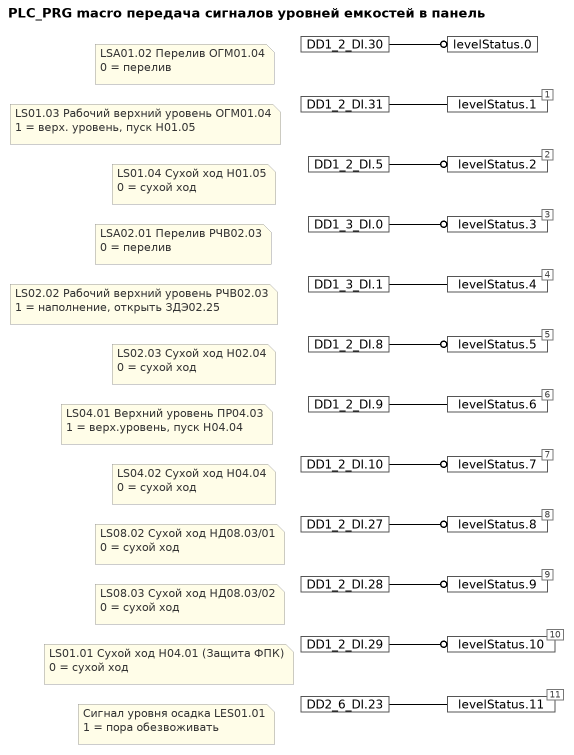
[picture p24: PLC_PRG macro передача сигналов уровней емкостей в панель (CFC)]
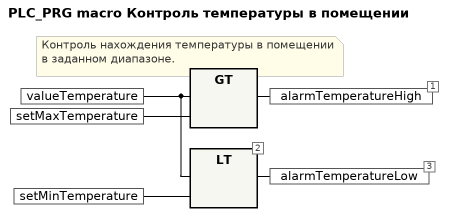
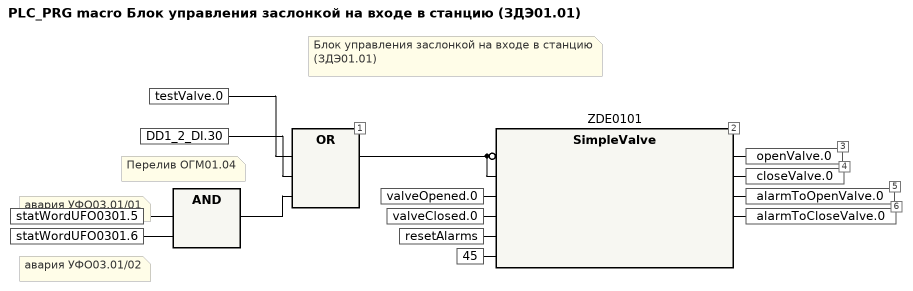
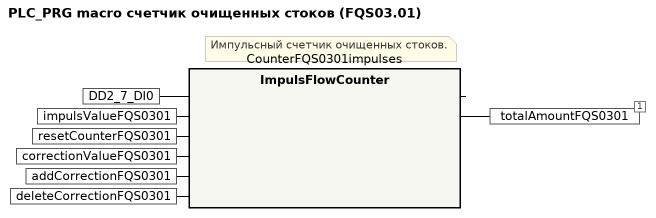
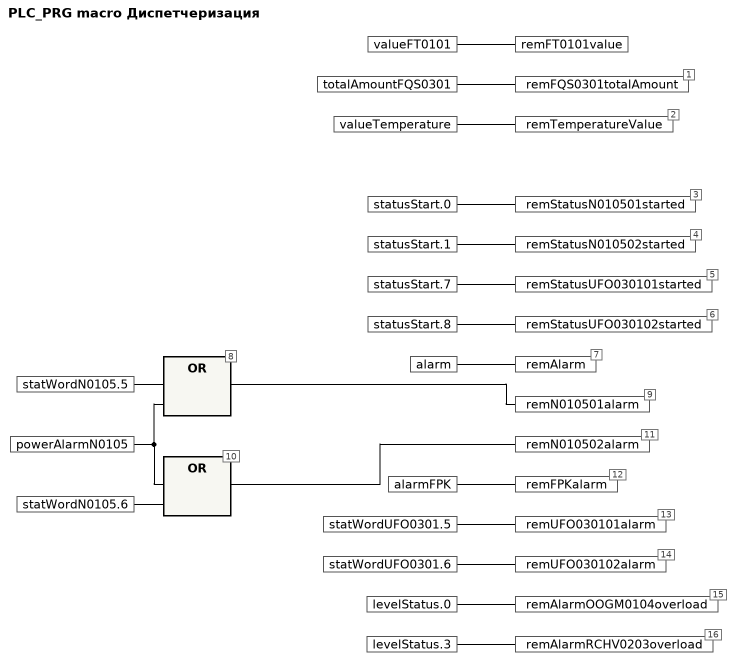
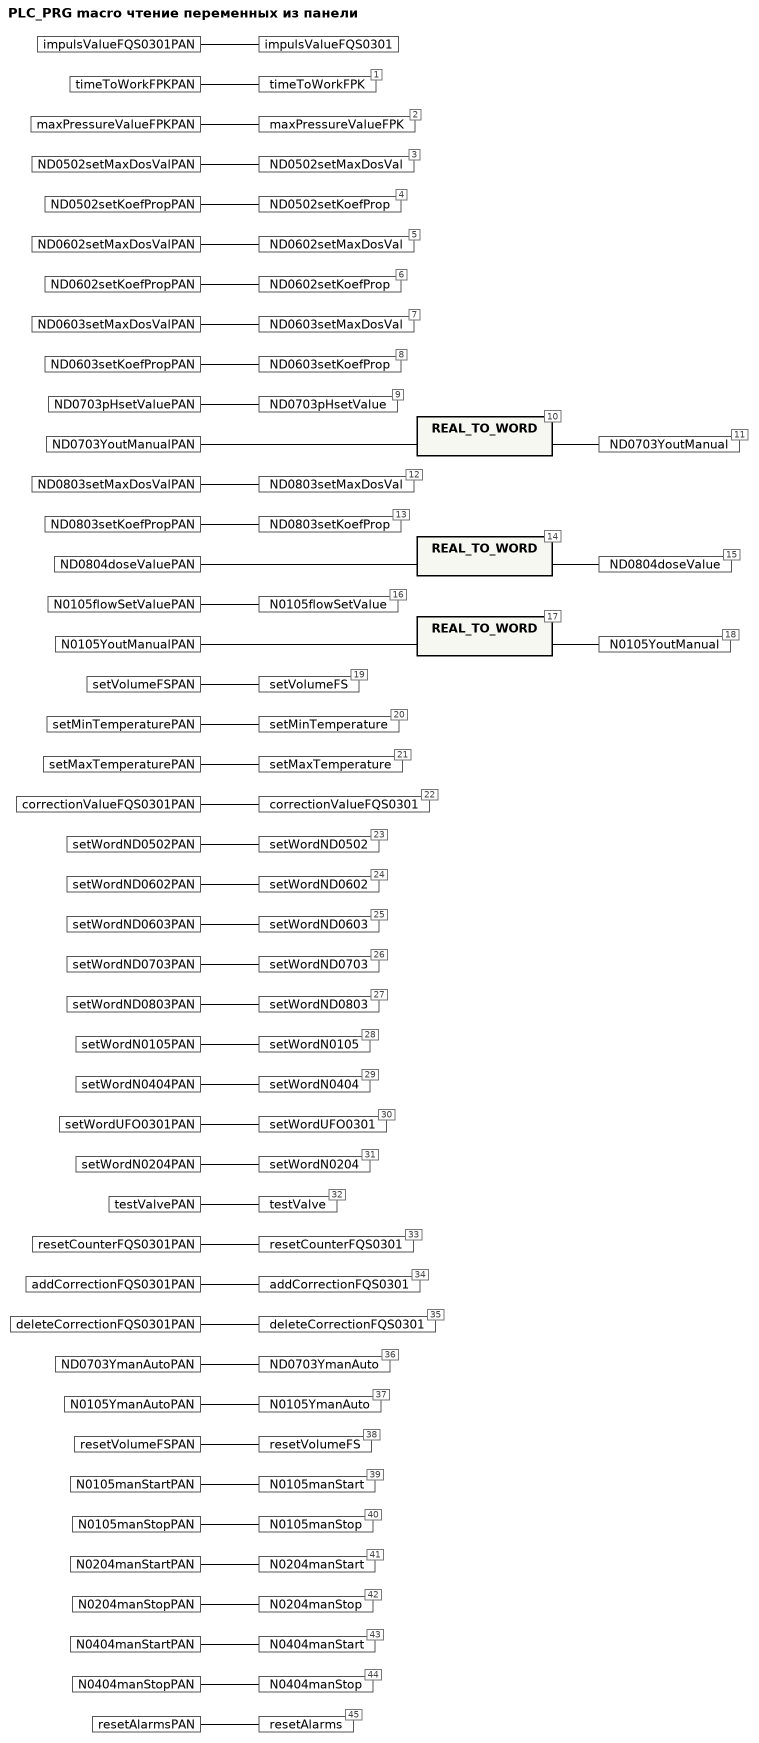
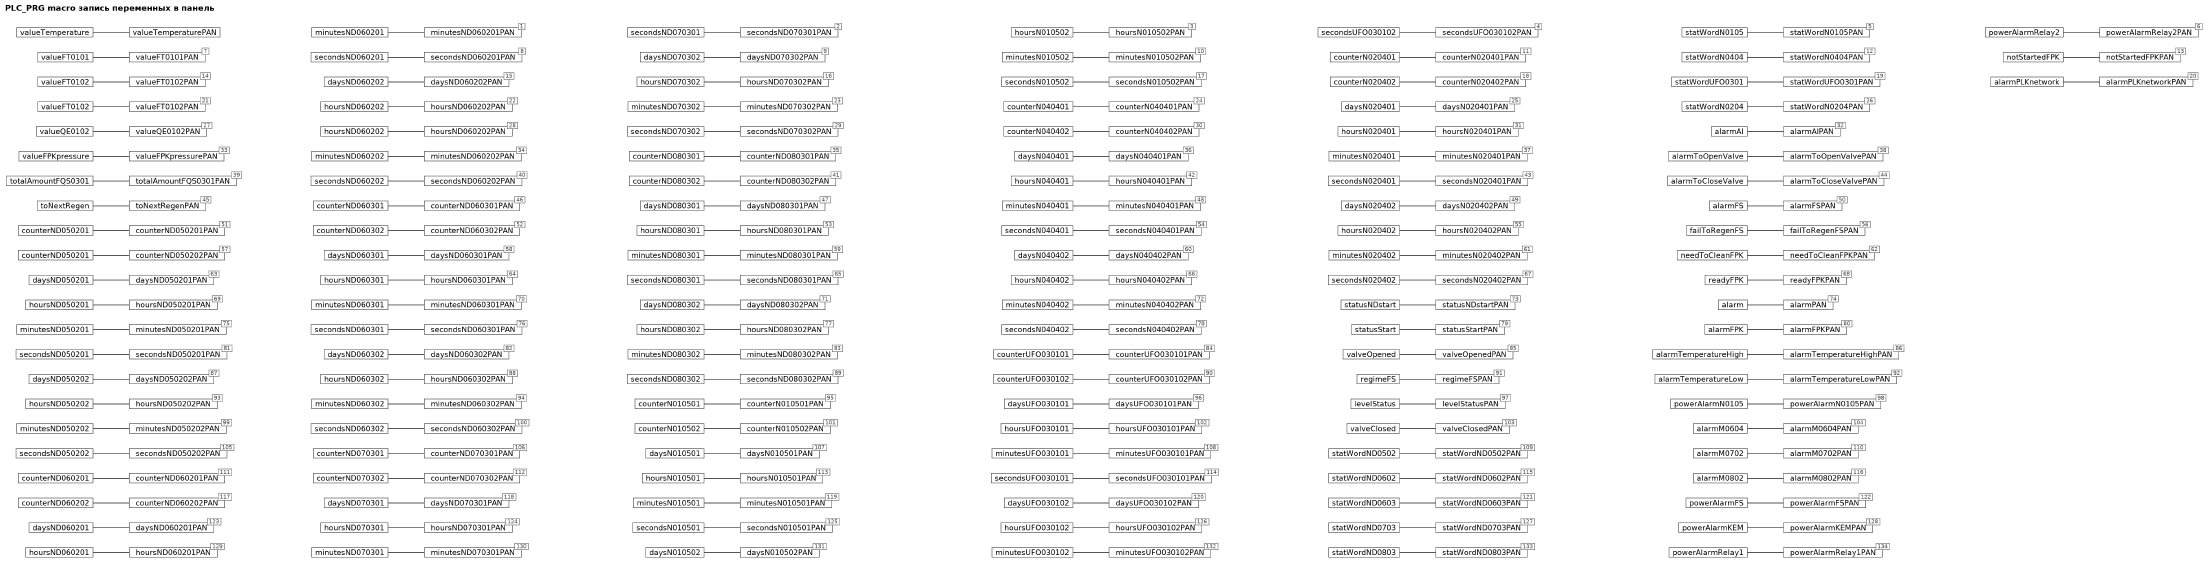
_CFC_ (* Continuous Function Chart, elements in execution order *)
#0 MACRO Блок задания всем режима по количеству включений при подаче питания()
	(* задать режим запуска УФО03.01 / по количеству включений *)
	(* задать режим запуска Н01.05 / по количеству включений *)
	(* задать режим запуска НД06.03 / по количеству включений *)
	(* задать режим запуска НД06.02 / по количеству включений *)
	(* задать режим запуска НД05.02 / по количеству включений *)
	(* задать режим запуска НД07.03 / по количеству включений *)
	(* задать режим запуска НД08.03 / по количеству включений *)
	(* задать режим запуска Н02.04 / по количеству включений *)
	(* задать режим запуска Н04.04 / по количеству включений *)
	#1 StartInitiBlock:R_TRIG(CLK: TRUE)
	#2 startInitializer <= #1.Q
	#3 setWordND0502.3 <= #1.Q
	#4 setWordND0602.3 <= #1.Q
	#5 setWordND0603.3 <= #1.Q
	#6 setWordND0703.3 <= #1.Q
	#7 setWordND0803.3 <= #1.Q
	#8 setWordN0105.3 <= #1.Q
	#9 setWordN0204.3 <= #1.Q
	#10 setWordN0404.3 <= #1.Q
	#11 setWordUFO0301.3 <= #1.Q
END_MACRO
#12 MACRO Управление доз.насосами НД05.02/01 и НД05.02/02()
	(* Управление доз.насосами НД05.02/01 и НД05.02/02 / пропорционально расходу по показаниям расходомера FT01.01 *)
	(* управление НД05.02/02 = 4...20мА *)
	(* управление НД05.02/01 = 4...20мА *)
	(* Если на входе sel = true, то нижнее значение, / иначе - посередине. Для того, чтобы при / выключении насоса не висело задание, / а сбрасывалось в ноль. *)
	(* Пуск НД05.02/01 *)
	(* Пуск НД05.02/02 *)
	#13 ND0502dosing:DosingPumpProportional(valueFT0101, -, ND0502setMaxDosVal, -, -, ND0502setKoefProp, -)
	#14 statWordND0502.0 <= #13.out 2
	#15 setWordND0502.0 <= #13.out 3
	#16 REAL_TO_WORD(#13.out 1)
	#17 ND0502manager:RichTwoPumpManager(setWordND0502.0, setWordND0502.1, setWordND0502.2, setWordND0502.3, setWordND0502.4, setWordND0502.5, setWordND0502.6, setWordND0502.7, setWordND0502.8, setWordND0502.9, setWordND0502.10, setWordND0502.11, resetAlarms, -, alarmND.0, alarmND.1)
	#18 statWordND0502.1 <= #17.out 1
	#19 statWordND0502.2 <= #17.out 2
	#20 statWordND0502.3 <= #17.out 3
	#21 statWordND0502.4 <= #17.out 4
	#22 counterND050201 <= #17.out 5
	#23 counterND050202 <= #17.out 6
	#24 daysND050201 <= #17.out 7
	#25 hoursND050201 <= #17.out 8
	#26 minutesND050201 <= #17.out 9
	#27 secondsND050201 <= #17.out 10
	#28 daysND050202 <= #17.out 11
	#29 hoursND050202 <= #17.out 12
	#30 minutesND050202 <= #17.out 13
	#31 secondsND050202 <= #17.out 14
	#32 statusNDstart.0 <= #17.out 15
	#33 DD1_1_DO.12 <= #17.out 15
	#34 DD1_1_DO.13 <= #17.out 16
	#35 statusNDstart.1 <= #17.out 16
	#36 statWordND0502.5 <= #17.out 19
	#37 statWordND0502.6 <= #17.out 20
	#38 SEL(#17.out 15, 4, #16)
	#39 lintrafoND050201:LIN_TRAFO(IN: #38, IN_MIN: 4, IN_MAX: 20, OUT_MIN: 0, OUT_MAX: 1000)
	#40 REAL_TO_WORD(#39.OUT)
	#41 DD1_4_AO0 <= #40
	#42 SEL(#17.out 16, 4, #16)
	#43 lintrafoND050202:LIN_TRAFO(IN: #42, IN_MIN: 4, IN_MAX: 20, OUT_MIN: 0, OUT_MAX: 1000)
	#44 REAL_TO_WORD(#43.OUT)
	#45 DD1_4_AO1 <= #44
END_MACRO
#46 MACRO Управление насосами Н01.05/01 и Н01.05/02()
	(* статус старт Н01.05/02 *)
	(* статус старт Н01.05/01 *)
	(* производительность для ЧРП Н01.05 *)
	(* командное слово для ЧРП Н01.05 *)
	(* Рабочий верхний уровень ОГМ01.04 *)
	(* Перелив ОГМ01.04 *)
	(* Сухой ход Н01.05 *)
	(* Термоконтакт Н01.05/02 *)
	(* Термоконтакт Н01.05/01 *)
	(* Авария привода Н01.05 (сигнал авария от ЧРП А1) *)
	(* Сигнал - ЧРП в режиме ПУСК, один из насосов работает. / Сигнал на лампы HL3-4 через доп.контакты КМ3.2 и КМ4.2 *)
	(* Питание Н01.05/01 (КМ4) *)
	(* Питание Н01.05/01 (КМ3) *)
	(* регулируем от 30 до 50Гц, чтобы не перегреть двигатель / 30Гц = 3258 *)
	(* 5430 = 50Гц *)
	(* Работа Н01.05 / Поддержание заданного расхода по FT01.02 / Пуск по верхнему рабочему уровню (LS01.03) или вручную с пульта / стоп по защите от сухого хода (LS01.04) или вручную с пульта *)
	(* Питание ЧРП Н01.05 (КМ2) *)
	(* слово состояния для ЧРП Н01.05 / сигнал - авария *)
	#47 linTrafoN0105:LIN_TRAFO(IN: N0105YoutManual, IN_MIN: 0, IN_MAX: 100, OUT_MIN: 0, OUT_MAX: 5430)
	#48 PID_ND0105:PID(ACTUAL: valueFT0102, SET_POINT: N0105flowSetValue, KP: 1, TN: 10, TV: 1, Y_MANUAL: #47.OUT, Y_OFFSET: 0, Y_MIN: 0, Y_MAX: 5430, MANUAL: N0105YmanAuto, RESET: #48.OVERFLOW)
	#49 LT(#48.Y, 3258)
	#50 SEL(#49, #48.Y, 3258)
	#51 REAL_TO_WORD(#50)
	#52 zad_rsN0105 <= #51
	#53 OR(DD1_2_DI.31, NOT DD1_2_DI.30, N0105manStart)
	#54 OR(NOT DD1_2_DI.5, N0105manStop)
	#55 rsTrigN0105:RS(SET: #53, RESET1: #54)
	#56 setWordN0105.0 <= #55.Q1
	#57 OR(DD1_2_DI.0, stat_wordN0105.3)
	#58 ND0105manager:TwoPumpOneDriveManager(setWordN0105.0, setWordN0105.1, setWordN0105.2, setWordN0105.3, setWordN0105.4, setWordN0105.5, setWordN0105.6, setWordN0105.7, setWordN0105.8, setWordN0105.9, setWordN0105.10, setWordN0105.11, resetAlarms, -, NOT DD1_2_DI.3, NOT DD1_2_DI.4, #57)
	#59 statWordN0105.1 <= #58.out 1
	#60 statWordN0105.2 <= #58.out 2
	#61 statWordN0105.3 <= #58.out 3
	#62 statWordN0105.4 <= #58.out 4
	#63 counterN010501 <= #58.out 5
	#64 counterN010502 <= #58.out 6
	#65 daysN010501 <= #58.out 7
	#66 hoursN010501 <= #58.out 8
	#67 minutesN010501 <= #58.out 9
	#68 secondsN010501 <= #58.out 10
	#69 daysN010502 <= #58.out 11
	#70 hoursN010502 <= #58.out 12
	#71 minutesN010502 <= #58.out 13
	#72 secondsN010502 <= #58.out 14
	#73 DD1_1_DO.0 <= #58.out 15
	#74 DD1_1_DO.1 <= #58.out 16
	#75 DD1_1_DO.2 <= #58.out 17
	#76 statWordN0105.5 <= #58.out 21
	#77 statWordN0105.6 <= #58.out 22
	#78 DD1_1_DO.3 <= #58.out 18
	#79 AND(DD1_1_DO.1, #58.out 18)
	#80 statusStart.0 <= #79
	#81 AND(#58.out 18, DD1_1_DO.2)
	#82 statusStart.1 <= #81
	#83 StartStopND0105:StartStopVFD(startStop: #58.out 18)
	#84 com_wordN0105 <= #83.commandWord
END_MACRO
#85 MACRO Сигналы "АВАРИЯ" от дозирующих насосов()
	(* Авария НД08.03/02 = stat_wordND080302.3 *)
	(* Авария НД08.03/01 = stat_wordND080301.3 *)
	(* Сигнал авария от физических выходов доз.насосов взят НЗ, т.е. / при замкнутом состоянии аварии нет. Если сигнал выдается только НО / (замкнуто = авария) - убрать инверсию здесь. / Сигнал авария по модбасу здесь взят как НО / т.е. false = норма, true - авария. *)
	(* Авария НД05.02/01 *)
	(* Авария НД05.02/02 *)
	(* Авария НД06.02/01 *)
	(* Авария НД06.02/02 *)
	(* Авария НД06.03/01 *)
	(* Авария НД06.03/02 *)
	(* Авария НД07.03/01 *)
	(* Авария НД07.03/02 *)
	(* Авария НД08.04 *)
	#86 alarmND.0 <= NOT DD1_2_DI.18
	#87 alarmND.1 <= NOT DD1_2_DI.19
	#88 alarmND.2 <= NOT DD1_2_DI.20
	#89 alarmND.3 <= NOT DD1_2_DI.21
	#90 alarmND.4 <= NOT DD1_2_DI.22
	#91 alarmND.5 <= NOT DD1_2_DI.23
	#92 alarmND.6 <= NOT DD1_2_DI.24
	#93 alarmND.7 <= NOT DD1_2_DI.25
	#94 alarmND.8 <= NOT DD2_6_DI.22
END_MACRO
#95 MACRO Управление доз.насосами НД06.02/01 и НД06.02/02()
	(* Управление доз.насосами НД06.02/01 и НД06.02/02 / пропорционально расходу по показаниям расходомера FT01.02 *)
	(* управление НД06.02/02 = 4...20мА *)
	(* управление НД06.02/01 = 4...20мА *)
	(* Если на входе sel = true, то нижнее значение, / иначе - посередине. Для того, чтобы при / выключении насоса не висело задание, / а сбрасывалось в ноль. *)
	(* Пуск НД06.02/01 *)
	(* Пуск НД06.02/02 *)
	#96 ND0602dosing:DosingPumpProportional(valueFT0102, -, ND0602setMaxDosVal, -, -, ND0602setKoefProp, -)
	#97 statWordND0602.0 <= #96.out 2
	#98 setWordND0602.0 <= #96.out 3
	#99 REAL_TO_WORD(#96.out 1)
	#100 ND0602manager:RichTwoPumpManager(setWordND0602.0, setWordND0602.1, setWordND0602.2, setWordND0602.3, setWordND0602.4, setWordND0602.5, setWordND0602.6, setWordND0602.7, setWordND0602.8, setWordND0602.9, setWordND0602.10, setWordND0602.11, resetAlarms, -, alarmND.2, alarmND.3)
	#101 statWordND0602.1 <= #100.out 1
	#102 statWordND0602.2 <= #100.out 2
	#103 statWordND0602.3 <= #100.out 3
	#104 statWordND0602.4 <= #100.out 4
	#105 counterND060201 <= #100.out 5
	#106 counterND060202 <= #100.out 6
	#107 daysND060201 <= #100.out 7
	#108 hoursND060201 <= #100.out 8
	#109 minutesND060201 <= #100.out 9
	#110 secondsND060201 <= #100.out 10
	#111 daysND060202 <= #100.out 11
	#112 hoursND060202 <= #100.out 12
	#113 minutesND060202 <= #100.out 13
	#114 secondsND060202 <= #100.out 14
	#115 statusNDstart.2 <= #100.out 15
	#116 DD1_1_DO.14 <= #100.out 15
	#117 DD1_1_DO.15 <= #100.out 16
	#118 statusNDstart.3 <= #100.out 16
	#119 statWordND0602.5 <= #100.out 19
	#120 statWordND0602.6 <= #100.out 20
	#121 SEL(#100.out 15, 4, #99)
	#122 lintrafoND060201:LIN_TRAFO(IN: #121, IN_MIN: 4, IN_MAX: 20, OUT_MIN: 0, OUT_MAX: 1000)
	#123 REAL_TO_WORD(#122.OUT)
	#124 DD1_4_AO2 <= #123
	#125 SEL(#100.out 16, 4, #99)
	#126 lintrafoND060202:LIN_TRAFO(IN: #125, IN_MIN: 4, IN_MAX: 20, OUT_MIN: 0, OUT_MAX: 1000)
	#127 REAL_TO_WORD(#126.OUT)
	#128 DD1_4_AO3 <= #127
END_MACRO
#129 MACRO Блок управления насосами Н02.04/01 и Н02.04/02()
	(* Минимум один из фильтров в режиме промывки *)
	(* Пуск Н02.04/02 *)
	(* Открыт минимум один из клапанов КЭМ *)
	(* Сухой ход Н02.04 / 1 = норма / 0 = сухой ход *)
	(* Авария Н02.04/02 *)
	(* Авария Н02.04/01 *)
	(* Пуск Н02.04/01 *)
	(* Блок управления насосами Н02.04/01 и Н02.04/02 / Включен, если хоть один из клапанов КЭМ открыт, / один из фильтров в промывке старт/стоп вручную (тест). *)
	(* автоматический пуск/стоп *)
	(* ручной пуск/стоп с защитой от сухого хода *)
	(* Сигнал на запуск насоса / согласно выбранному режиму *)
	#130 WORD_TO_BOOL(openedKEM)
	#131 WORD_TO_BOOL(regimeFS)
	#132 OR(#130, #131)
	#133 AND(#132, DD1_2_DI.8)
	#134 OR(NOT DD1_2_DI.8, N0204manStop)
	#135 N0204startTrig:RS(SET: N0204manStart, RESET1: #134)
	#136 OR(#133, #135.Q1)
	#137 setWordN0204.0 <= #136
	#138 N0204manager:RichTwoPumpManager(setWordN0204.0, setWordN0204.1, setWordN0204.2, setWordN0204.3, setWordN0204.4, setWordN0204.5, setWordN0204.6, setWordN0204.7, setWordN0204.8, setWordN0204.9, setWordN0204.10, setWordN0204.11, resetAlarms, -, DD1_2_DI.6, DD1_2_DI.7)
	#139 statWordN0204.1 <= #138.out 1
	#140 statWordN0204.2 <= #138.out 2
	#141 statWordN0204.3 <= #138.out 3
	#142 statWordN0204.4 <= #138.out 4
	#143 counterN020401 <= #138.out 5
	#144 counterN020402 <= #138.out 6
	#145 daysN020401 <= #138.out 7
	#146 hoursN020401 <= #138.out 8
	#147 minutesN020401 <= #138.out 9
	#148 daysN020402 <= #138.out 11
	#149 hoursN020402 <= #138.out 12
	#150 minutesN020402 <= #138.out 13
	#151 statusStart.2 <= #138.out 15
	#152 secondsN020402 <= #138.out 14
	#153 DD1_1_DO.4 <= #138.out 15
	#154 DD1_1_DO.5 <= #138.out 16
	#155 statusStart.3 <= #138.out 16
	#156 statWordN0204.5 <= #138.out 19
	#157 statWordN0204.6 <= #138.out 20
END_MACRO
#158 MACRO Блок сбора всех аварий и выдачи одной общей()
	(* Контроль состояния сети ПЛК, задержка выдачи сигнала = 20 сек. / Контроль обрыва в сети (модуль отсоединен, или модуль в аварии. *)
	(* ошибка блоков дозирования / (неправильно выставлены / параметры в настройках) *)
	(* лампа Авария / (щит-1) *)
	(* Авария питания ЧРП А1 (автомат ЧРП выключен) *)
	(* Перелив ОГМ01.04 (отстойник) *)
	(* Перелив РЧВ02.03 *)
	(* Авария М08.02 (УПФ) *)
	(* Авария М07.02 (УПЩ) *)
	(* Авария М06.04 (УПК) *)
	(* Авария питания управляющих клапанов фильтров *)
	(* Авария питания клапанов КЭМ *)
	(* Авария питания K, KM, HL щит1 *)
	(* Авария питания реле щита 2 *)
	(* Авария фильтр-пресса (ФП) *)
	#159 WORD_TO_BOOL(alarmAI)
	#160 DWORD_TO_BOOL(alarmToOpenValve)
	#161 DWORD_TO_BOOL(alarmToCloseValve)
	#162 WORD_TO_BOOL(alarmFS)
	#163 WORD_TO_BOOL(failToRegenFS)
	#164 EQ(lastError, 0)
	#165 alarmPLKnetworkDelay:TOF(IN: #164, PT: T#20s)
	#166 NOT(#165.Q)
	#167 alarmPLKnetwork <= #166
	#168 OR(#159, alarmTemperatureHigh, alarmTemperatureLow, statWordND0502.5, statWordND0502.6, statWordND0602.5, statWordND0602.6, statWordND0603.5, statWordND0603.6, statWordND0703.5, statWordND0703.6, statWordND0803.5, statWordND0803.6, powerAlarmN0105, statWordN0105.5, statWordN0105.6, levelStatus.0, statWordN0204.5, statWordN0204.6, statWordN0404.5, statWordN0404.6, #160, #161, alarmM0604, alarmM0702, alarmM0802, powerAlarmFS, levelStatus.3, powerAlarmKEM, powerAlarmRelay1, powerAlarmRelay2, alarmFPK, notStartedFPK, #162, #163, statWordUFO0301.5, statWordUFO0301.6, statWordND0502.0, statWordND0602.0, statWordND0603.0, statWordND0803.0, alarmND.8, #166)
	#169 alarm <= #168
	#170 DD1_1_DO.8 <= #168
	#171 powerAlarmN0105 <= DD1_2_DI.2
	#172 alarmM0604 <= NOT DD1_2_DI.15
	#173 alarmM0702 <= NOT DD1_2_DI.16
	#174 alarmM0802 <= NOT DD1_2_DI.17
	#175 powerAlarmFS <= NOT DD1_2_DI.26
	#176 powerAlarmKEM <= NOT DD1_3_DI.2
	#177 powerAlarmRelay1 <= NOT DD1_2_DI.1
	#178 powerAlarmRelay2 <= NOT DD2_4_DI.0
	#179 alarmFPK <= DD2_6_DI.21
END_MACRO
#180 MACRO Управление доз.насосами НД06.03/01 и НД06.03/02()
	(* Управление доз.насосами НД06.03/01 и НД06.03/02 / пропорционально расходу по показаниям расходомера FT01.01 *)
	(* управление НД06.03/02 = 4...20мА *)
	(* управление НД06.03/01 = 4...20мА *)
	(* Если на входе sel = true, то нижнее значение, / иначе - посередине. Для того, чтобы при / выключении насоса не висело задание, / а сбрасывалось в ноль. *)
	(* Пуск НД06.03/01 *)
	(* Пуск НД06.03/02 *)
	#181 ND0603dosing:DosingPumpProportional(valueFT0101, -, ND0603setMaxDosVal, -, -, ND0603setKoefProp, -)
	#182 statWordND0603.0 <= #181.out 2
	#183 setWordND0603.0 <= #181.out 3
	#184 REAL_TO_WORD(#181.out 1)
	#185 ND0603manager:RichTwoPumpManager(setWordND0603.0, setWordND0603.1, setWordND0603.2, setWordND0603.3, setWordND0603.4, setWordND0603.5, setWordND0603.6, setWordND0603.7, setWordND0603.8, setWordND0603.9, setWordND0603.10, setWordND0603.11, resetAlarms, -, alarmND.4, alarmND.5)
	#186 statWordND0603.1 <= #185.out 1
	#187 statWordND0603.2 <= #185.out 2
	#188 statWordND0603.3 <= #185.out 3
	#189 statWordND0603.4 <= #185.out 4
	#190 counterND060301 <= #185.out 5
	#191 counterND060302 <= #185.out 6
	#192 daysND060301 <= #185.out 7
	#193 hoursND060301 <= #185.out 8
	#194 minutesND060301 <= #185.out 9
	#195 secondsND060301 <= #185.out 10
	#196 daysND060302 <= #185.out 11
	#197 hoursND060302 <= #185.out 12
	#198 minutesND060302 <= #185.out 13
	#199 secondsND060302 <= #185.out 14
	#200 statusNDstart.4 <= #185.out 15
	#201 DD1_1_DO.16 <= #185.out 15
	#202 DD1_1_DO.17 <= #185.out 16
	#203 statusNDstart.5 <= #185.out 16
	#204 statWordND0603.5 <= #185.out 19
	#205 statWordND0603.6 <= #185.out 20
	#206 SEL(#185.out 15, 4, #184)
	#207 linrtafoND060301:LIN_TRAFO(IN: #206, IN_MIN: 4, IN_MAX: 20, OUT_MIN: 0, OUT_MAX: 1000)
	#208 REAL_TO_WORD(#207.OUT)
	#209 DD1_4_AO4 <= #208
	#210 SEL(#185.out 16, 4, #184)
	#211 linrtafoND060302:LIN_TRAFO(IN: #210, IN_MIN: 4, IN_MAX: 20, OUT_MIN: 0, OUT_MAX: 1000)
	#212 REAL_TO_WORD(#211.OUT)
	#213 DD1_4_AO5 <= #212
END_MACRO
#214 MACRO Блок управления насосами Н04.04/01 и Н04.04/02()
	(* Сухой ход Н04.04 / 1 = норма / 0 = сухой ход *)
	(* Блок управления насосами Н04.04/01 и Н04.04/02 / Дренажные насосы. Работа по поплавкам (LS04.01 и LS04.02) или пуск вручную (тест). *)
	(* автоматический пуск/стоп *)
	(* ручной пуск/стоп с защитой от сухого хода *)
	(* Сигнал на запуск насоса / согласно выбранному режиму *)
	(* Пуск Н04.04/01 *)
	(* Пуск Н04.04/02 *)
	(* Верхний уровень ПР04.03 *)
	(* Авария Н04.04/01 *)
	(* Авария Н04.04/02 *)
	#215 AND(DD1_2_DI.9, DD1_2_DI.10)
	#216 OR(NOT DD1_2_DI.10, N0404manStop)
	#217 N0404startTrig:RS(SET: N0404manStart, RESET1: #216)
	#218 OR(#215, #217.Q1)
	#219 setWordN0404.0 <= #218
	#220 N0404manager:RichTwoPumpManager(setWordN0404.0, setWordN0404.1, setWordN0404.2, setWordN0404.3, setWordN0404.4, setWordN0404.5, setWordN0404.6, setWordN0404.7, setWordN0404.8, setWordN0404.9, setWordN0404.10, setWordN0404.11, resetAlarms, -, DD1_2_DI.11, DD1_2_DI.12)
	#221 statWordN0404.1 <= #220.out 1
	#222 statWordN0404.2 <= #220.out 2
	#223 statWordN0404.3 <= #220.out 3
	#224 statWordN0404.4 <= #220.out 4
	#225 counterN040401 <= #220.out 5
	#226 counterN040402 <= #220.out 6
	#227 daysN040401 <= #220.out 7
	#228 hoursN040401 <= #220.out 8
	#229 minutesN040401 <= #220.out 9
	#230 secondsN040401 <= #220.out 10
	#231 daysN040402 <= #220.out 11
	#232 hoursN040402 <= #220.out 12
	#233 minutesN040402 <= #220.out 13
	#234 DD1_1_DO.6 <= #220.out 15
	#235 secondsN040402 <= #220.out 14
	#236 statusStart.4 <= #220.out 15
	#237 statusStart.5 <= #220.out 16
	#238 DD1_1_DO.7 <= #220.out 16
	#239 statWordN0404.5 <= #220.out 19
	#240 statWordN0404.6 <= #220.out 20
END_MACRO
#241 MACRO AI PLC (блок обработки аналоговых входов)()
	(* Здесь принимаем сигнал от входа ПЛК, в нем должно быть выставлен диапазон 0...20 / Задаем максимальное и минимальное значение для измеряемой величины при 4 и 20мА на датчике. *)
	(* рН *)
	(* рН *)
	(* бар *)
	(* куб.м./час *)
	(* куб.м./час *)
	(* Давление на входе / в фильтр-пресс *)
	(* рН-ОВП метр QE01.02 *)
	(* рН-ОВП метр QE01.01 *)
	(* Расходомер FT01.02 *)
	(* град.С *)
	(* Расходомер FT01.01 *)
	(* датчик температуры / в помещении TT01 *)
	(* Авария датчика температуры *)
	(* Авария расходомера FT01.01 *)
	(* Авария расходомера FT01.02 *)
	(* Авария рН-метра QE01.01 *)
	(* Авария рН-метра QE01.02 *)
	(* Авария входа приема показаний / давления на входе в фильтр *)
	#242 ControlAI0:ControlAI(DD2_7_AI0, -40, 80)
	#243 valueTemperature <= #242.out 1
	#244 alarmAI.0 <= #242.out 2
	#245 ControlAI1:ControlAI(DD2_7_AI1, -, 600)
	#246 valueFT0101 <= #245.out 1
	#247 alarmAI.1 <= #245.out 2
	#248 ControlAI2:ControlAI(DD2_7_AI2, -, 600)
	#249 valueFT0102 <= #248.out 1
	#250 alarmAI.2 <= #248.out 2
	#251 ControlAI3:ControlAI(DD2_7_AI3, -, 14)
	#252 valueQE0101 <= #251.out 1
	#253 alarmAI.3 <= #251.out 2
	#254 ControlAI4:ControlAI(DD2_7_AI4, -, 14)
	#255 valueQE0102 <= #254.out 1
	#256 alarmAI.4 <= #254.out 2
	#257 ControlAI5:ControlAI(DD2_7_AI5, -, 16)
	#258 valueFPKpressure <= #257.out 1
	#259 alarmAI.5 <= #257.out 2
END_MACRO
#260 MACRO Управление доз.насосами НД07.03/01 и НД07.03/02()
	(* коэф. P *)
	(* Пуск, если по FT01.01 / расход >= 10 куб.метров *)
	(* Управление доз.насосами НД07.03/01 и НД07.03/02 / поддержание заданного уровня рН по показаниям QE01.01 *)
	(* управление НД07.03/02 = 4...20мА *)
	(* управление НД07.03/01 = 4...20мА *)
	(* Если на входе sel = true, то нижнее значение, / иначе - посередине. Для того, чтобы при / выключении насоса не висело задание, / а сбрасывалось в ноль. *)
	(* Пуск НД07.03/01 *)
	(* Пуск НД07.03/02 *)
	(* коэф. I *)
	(* коэф. D *)
	(* Y при аварии *)
	#261 manYoutND0703:LIN_TRAFO(IN: ND0703YoutManual, IN_MIN: 0, IN_MAX: 100, OUT_MIN: 4, OUT_MAX: 20)
	#262 ND0703pidReg:PID(ACTUAL: valueQE0101, SET_POINT: ND0703pHsetValue, KP: 1, TN: 10, TV: 1, Y_MANUAL: #261.OUT, Y_OFFSET: 12, Y_MIN: 4, Y_MAX: 20, MANUAL: ND0703YmanAuto, RESET: #262.OVERFLOW)
	#263 REAL_TO_WORD(#262.Y)
	#264 GE(valueFT0101, 10)
	#265 ND0703manager:RichTwoPumpManager(#264, setWordND0703.1, setWordND0703.2, setWordND0703.3, setWordND0703.4, setWordND0703.5, setWordND0703.6, setWordND0703.7, setWordND0703.8, setWordND0703.9, setWordND0703.10, setWordND0703.11, resetAlarms, -, alarmND.6, alarmND.7)
	#266 statWordND0703.1 <= #265.out 1
	#267 statWordND0703.2 <= #265.out 2
	#268 statWordND0703.3 <= #265.out 3
	#269 statWordND0703.4 <= #265.out 4
	#270 counterND070301 <= #265.out 5
	#271 counterND070302 <= #265.out 6
	#272 daysND070301 <= #265.out 7
	#273 hoursND070301 <= #265.out 8
	#274 minutesND070301 <= #265.out 9
	#275 secondsND070301 <= #265.out 10
	#276 daysND070302 <= #265.out 11
	#277 hoursND070302 <= #265.out 12
	#278 minutesND070302 <= #265.out 13
	#279 secondsND070302 <= #265.out 14
	#280 statusNDstart.6 <= #265.out 15
	#281 DD1_1_DO.18 <= #265.out 15
	#282 DD1_1_DO.19 <= #265.out 16
	#283 statusNDstart.7 <= #265.out 16
	#284 statWordND0703.5 <= #265.out 19
	#285 statWordND0703.6 <= #265.out 20
	#286 SEL(#265.out 15, 4, #263)
	#287 lintrafoND070301:LIN_TRAFO(IN: #286, IN_MIN: 4, IN_MAX: 20, OUT_MIN: 0, OUT_MAX: 1000)
	#288 REAL_TO_WORD(#287.OUT)
	#289 DD1_4_AO6 <= #288
	#290 SEL(#265.out 16, 4, #263)
	#291 lintrafoND070302:LIN_TRAFO(IN: #290, IN_MIN: 4, IN_MAX: 20, OUT_MIN: 0, OUT_MAX: 1000)
	#292 REAL_TO_WORD(#291.OUT)
	#293 DD1_4_AO7 <= #292
END_MACRO
#294 MACRO Алгоритм работы фильтр-пресса и КШЭ04.01()
	(* Тестировать заслонку. / 1 = открыть, / 0 = закрыть *)
	(* Фильтр-пресс надо почистить *)
	(* Алгоритм работы фильтр-пресса и КШЭ04.01 *)
	(* Время работы ФПК после спада сигнала уровня осадка / Если переменную не использовать в панели, то 900 сек (15 мин). *)
	(* авария входа датчика давления *)
	(* Старт обезвоживания на ФПК *)
	(* Статус ФП готов к приему осадка *)
	(* Подающий насос ФП работает *)
	(* Авария фильтр-пресса (ФП) *)
	(* Сигнал уровня осадка LES01.01 / 1 = пора обезвоживать *)
	(* LS01.01 сух.ход Н04.01 (ФПК), 0 = авария. *)
	(* Условие сброса сигнала о необходимости почистить фильтр: / 1. пропал сигнал готовности ФПК / 2. Появился сигнал готовности ФПК / это значит: плиты раздвигали, наверное, чистили, сдвигали. *)
	(* КШЭ04.01 не открылась *)
	(* блок управления заслонкой КШЭ04.01 *)
	(* время на открытие/закрытие / заслонки, секунд. *)
	#295 statusStart.6 <= DD2_6_DI.20
	#296 readyFPK <= DD2_6_DI.19
	#297 WORD_TO_TIME(timeToWorkFPK)
	#298 MUL(#297, 1000)
	#299 FPKstopTimer:TOF(IN: DD2_6_DI.23, PT: #298)
	#300 FPKstopFtrig:F_TRIG(CLK: #299.Q)
	#301 OR(#300.Q, alarmAI.5, DD2_6_DI.21, NOT DD1_2_DI.29, needToCleanFPK, alarmToOpenValve.28, NOT DD2_6_DI.19)
	#302 FPKstartTrig:RS(SET: DD2_6_DI.23, RESET1: #301)
	#303 DD2_2_DO.26 <= #302.Q1
	#304 notStartedFPKtimer:TON(IN: #302.Q1, PT: T#300s)
	#305 AND(#304.Q, NOT DD2_6_DI.20)
	#306 notStartedFPK <= #305
	#307 OR(#302.Q1, testValve.28)
	#308 valveKSHE0401:SimpleValve(#307, NOT #307, valveOpened.28, valveClosed.28, resetAlarms, 45)
	#309 openValve.28 <= #308.out 1
	#310 closeValve.28 <= #308.out 2
	#311 alarmToOpenValve.28 <= #308.out 3
	#312 alarmToCloseValve.28 <= #308.out 4
	#313 GE(valueFPKpressure, maxPressureValueFPK)
	#314 readyFPKrTrig:R_TRIG(CLK: DD2_6_DI.19)
	#315 needToClleanFPKtrig:RS(SET: #313, RESET1: #314.Q)
	#316 needToCleanFPK <= #315.Q1
END_MACRO
#317 MACRO Обмен сигналами с управляющими клапанами фильтров()
	(* Подача управляющего сигнала в клапан фильтра. / 0 = нет сигнала; / 1 = начать промывку (регенерацию) *)
	(* Сигнал от управляющего клапана фильтра / о текущем режиме: / 0 = фильтрация; / 1 = промывка. *)
	(* Сигнал авария от управляющего клапана / фильтра. Исходный сигнал: 0 = авария, 1 = норма. / В общую переменную alarmFS / записывается инвертированно: 0 = норма, 1 = авария. *)
	(* ФС02.01/01 *)
	(* ФС02.01/02 *)
	(* ФС02.01/03 *)
	(* ФС02.01/04 *)
	(* ФС02.01/05 *)
	(* ФС02.01/06 *)
	(* ФС02.02/01 *)
	(* ФС02.02/02 *)
	(* ФС02.02/03 *)
	(* ФС02.02/04 *)
	(* ФС02.02/05 *)
	(* ФС02.02/06 *)
	#318 DD2_2_DO.28 <= setRegimeFS.0
	#319 regimeFS.0 <= DD2_5_DI.27
	#320 alarmFS.0 <= NOT DD2_5_DI.28
	#321 DD2_2_DO.29 <= setRegimeFS.1
	#322 regimeFS.1 <= DD2_5_DI.29
	#323 alarmFS.1 <= NOT DD2_5_DI.30
	#324 DD2_2_DO.30 <= setRegimeFS.2
	#325 regimeFS.2 <= DD2_5_DI.31
	#326 alarmFS.2 <= NOT DD2_6_DI.0
	#327 DD2_2_DO.31 <= setRegimeFS.3
	#328 regimeFS.3 <= DD2_6_DI.1
	#329 alarmFS.3 <= NOT DD2_6_DI.2
	#330 DD2_3_DO.0 <= setRegimeFS.4
	#331 regimeFS.4 <= DD2_6_DI.3
	#332 alarmFS.4 <= NOT DD2_6_DI.4
	#333 DD2_3_DO.1 <= setRegimeFS.5
	#334 regimeFS.5 <= DD2_6_DI.5
	#335 alarmFS.5 <= NOT DD2_6_DI.6
	#336 DD2_3_DO.2 <= setRegimeFS.6
	#337 regimeFS.6 <= DD2_6_DI.7
	#338 alarmFS.6 <= NOT DD2_6_DI.8
	#339 DD2_3_DO.3 <= setRegimeFS.7
	#340 regimeFS.7 <= DD2_6_DI.9
	#341 alarmFS.7 <= NOT DD2_6_DI.10
	#342 DD2_3_DO.4 <= setRegimeFS.8
	#343 regimeFS.8 <= DD2_6_DI.11
	#344 alarmFS.8 <= NOT DD2_6_DI.12
	#345 DD2_3_DO.5 <= setRegimeFS.9
	#346 regimeFS.9 <= DD2_6_DI.13
	#347 alarmFS.9 <= NOT DD2_6_DI.14
	#348 DD2_3_DO.6 <= setRegimeFS.10
	#349 regimeFS.10 <= DD2_6_DI.15
	#350 alarmFS.10 <= NOT DD2_6_DI.16
	#351 DD2_3_DO.7 <= setRegimeFS.11
	#352 regimeFS.11 <= DD2_6_DI.17
	#353 alarmFS.11 <= NOT DD2_6_DI.18
END_MACRO
#354 MACRO Управление доз.насосами НД08.03/01 и НД08.03/02()
	(* авария питания ЧРП или реле ЧРП *)
	(* авария ЧРП по модбас *)
	(* сухой ход НД08.03/01 *)
	(* авария питания ЧРП или реле ЧРП *)
	(* авария ЧРП по модбас *)
	(* Управление доз.насосами НД08.03/01 и НД08.03/02 / пропорционально расходу по показаниям расходомера FT01.01 *)
	(* управление НД08.03/02 = 30...50Гц *)
	(* управление НД08.03/01 = 30...50Гц *)
	(* Если на входе sel = true, то нижнее значение, / иначе - посередине. Для того, чтобы при / выключении насоса не висело задание, / а сбрасывалось в ноль. *)
	(* Пуск НД08.03/01 *)
	(* Пуск НД08.03/02 *)
	(* клемма 29, ТК эл.дв. если есть *)
	(* клемма 29, ТК эл.дв. если есть *)
	(* 5430 = 50Гц, *)
	(* регулируем от 30 до 50Гц, чтобы не перегреть двигатель / 30 = 3258. *)
	(* сухой ход НД08.03/02 *)
	(* сухой ход НД08.03/01 *)
	(* сухой ход НД08.03/02 *)
	#355 ND0803dosing:DosingPumpProportional(valueFT0101, -, ND0803setMaxDosVal, -, -, ND0803setKoefProp, -)
	#356 statWordND0803.0 <= #355.out 2
	#357 setWordND0803.0 <= #355.out 3
	#358 linTrafoND0803:LIN_TRAFO(IN: #355.out 1, IN_MIN: 4, IN_MAX: 20, OUT_MIN: 0, OUT_MAX: 5430)
	#359 LT(#358.OUT, 3258)
	#360 SEL(#359, #358.OUT, 3258)
	#361 REAL_TO_WORD(#360)
	#362 WORD_TO_BOOL(di29ND080301)
	#363 OR(stat_wordND080301.3, NOT DD1_2_DI.13, NOT DD1_2_DI.27, NOT DD1_2_DI.28, NOT #362)
	#364 WORD_TO_BOOL(di29ND080302)
	#365 OR(stat_wordND080301.3, NOT DD1_2_DI.13, NOT DD1_2_DI.27, NOT DD1_2_DI.28, NOT #364)
	#366 ND0803manager:RichTwoPumpManager(setWordND0803.0, setWordND0803.1, setWordND0803.2, setWordND0803.3, setWordND0803.4, setWordND0803.5, setWordND0803.6, setWordND0803.7, setWordND0803.8, setWordND0803.9, setWordND0803.10, setWordND0803.11, resetAlarms, -, #363, #365)
	#367 statWordND0803.1 <= #366.out 1
	#368 statWordND0803.2 <= #366.out 2
	#369 statWordND0803.3 <= #366.out 3
	#370 statWordND0803.4 <= #366.out 4
	#371 counterND080301 <= #366.out 5
	#372 counterND080302 <= #366.out 6
	#373 daysND080301 <= #366.out 7
	#374 hoursND080301 <= #366.out 8
	#375 statusNDstart.8 <= #366.out 15
	#376 minutesND080301 <= #366.out 9
	#377 secondsND080301 <= #366.out 10
	#378 daysND080302 <= #366.out 11
	#379 hoursND080302 <= #366.out 12
	#380 minutesND080302 <= #366.out 13
	#381 secondsND080302 <= #366.out 14
	#382 statusNDstart.9 <= #366.out 16
	#383 statWordND0803.5 <= #366.out 19
	#384 statWordND0803.6 <= #366.out 20
	#385 SEL(#366.out 15, 0, #361)
	#386 zad_rsND080301 <= #385
	#387 SEL(#366.out 16, 0, #361)
	#388 zad_rsND080302 <= #387
	#389 startStopND080301:StartStopVFD(startStop: #366.out 15)
	#390 com_wordND080301 <= #389.commandWord
	#391 startStopND080302:StartStopVFD(startStop: #366.out 16)
	#392 com_wordND080302 <= #391.commandWord
END_MACRO
#393 MACRO Наполнение РЧВ02.23, заслонка ЗДЭ02.25()
	(* Наполнение РЧВ02.23, заслонка ЗДЭ02.25 *)
	(* Рабочий верхний уровень РЧВ02.03 / 0 = верхний уровень достигнут *)
	(* Перелив РЧВ02.03 / 0 = перелив *)
	(* время открытия/закрытия, сек. *)
	#394 OR(testValve.25, DD1_3_DI.1)
	#395 AND(DD1_3_DI.0, #394)
	#396 valveZDE0225:SimpleValve(#395, NOT #395, valveOpened.25, valveClosed.25, resetAlarms, 45)
	#397 openValve.25 <= #396.out 1
	#398 closeValve.25 <= #396.out 2
	#399 alarmToOpenValve.25 <= #396.out 3
	#400 alarmToCloseValve.25 <= #396.out 4
END_MACRO
#401 MACRO сигналы об открытии клапанов КЭМ()
	(* открыт КЭМ05.01 *)
	(* клапанаы наполнения реагентных емкостей, / сигнал используется для включения подачи насосами Н02.04 *)
	(* открыт КЭМ06.01 *)
	(* открыт КЭМ07.01 *)
	(* открыт КЭМ08.01 *)
	#402 openedKEM.0 <= DD1_3_DI.3
	#403 openedKEM.1 <= DD1_3_DI.4
	#404 openedKEM.2 <= DD1_3_DI.5
	#405 openedKEM.3 <= DD1_3_DI.6
END_MACRO
#406 MACRO управление дозирующим насосом НД08.04.()
	(* Подающий насос ФП работает *)
	(* Пуск/стоп НД08.04 *)
	(* управление дозирующим насосом НД08.04. / Работа с заранее заданной производительностью 0...100% / при работе подающего насоса ФП. *)
	(* Авария НД08.04 *)
	(* управление НД08.04 = 4...20мА *)
	(* Если на входе sel = true, то нижнее значение, / иначе - посередине. Для того, чтобы при / выключении насоса не висело задание, / а сбрасывалось в ноль. *)
	#407 AND(DD2_6_DI.20, NOT alarmND.8)
	#408 statusNDstart.10 <= #407
	#409 DD2_2_DO.27 <= #407
	#410 WORD_TO_REAL(ND0804doseValue)
	#411 linTrafND0804:LIN_TRAFO(IN: #410, IN_MIN: 0, IN_MAX: 100, OUT_MIN: 4, OUT_MAX: 20)
	#412 SEL(#407, 0, #411.OUT)
	#413 DD2_7_AO0 <= #412
END_MACRO
#414 MACRO блок управления очередью промывки/регенерации()
	(* фильтрация: ЗДЭ02.01, промывка: ЗДЭ02.07 *)
	(* фильтрация: ЗДЭ02.13, промывка: ЗДЭ02.19 *)
	(* фильтрация: ЗДЭ02.02, промывка: ЗДЭ02.08 *)
	(* фильтрация: ЗДЭ02.14, промывка: ЗДЭ02.20 *)
	(* фильтрация: ЗДЭ02.03, промывка: ЗДЭ02.09 *)
	(* фильтрация: ЗДЭ02.15, промывка: ЗДЭ02.21 *)
	(* фильтрация: ЗДЭ02.04, промывка: ЗДЭ02.10 *)
	(* фильтрация: ЗДЭ02.16, промывка: ЗДЭ02.22 *)
	(* фильтрация: ЗДЭ02.05, промывка: ЗДЭ02.11 *)
	(* фильтрация: ЗДЭ02.17, промывка: ЗДЭ02.23 *)
	(* фильтрация: ЗДЭ02.06, промывка: ЗДЭ02.12 *)
	(* фильтрация: ЗДЭ02.18, промывка: ЗДЭ02.24 *)
	(* Блок управления промывкой/фильтрацией. / valueFT0102 - данные расходомера FT01.02 / setVolumeFS - задание объема до промывки / resetVolumeFS - ручной сброс счетчика / totalAmountFS - объем стоков после последней промывки / Когда объем стоков сравняется с заданием счетчик сбрасывается / и выдает импульс в очередь фильтров на промывку. / В очереди на промывку встает фильтр, в котором нет аварии и / отметки, что он уже прорегенерировал. / Когда промоется последний фильтр, сбрасываются все отметки / о промытости и очередь начинается с начала. *)
	(* счетчик стоков до промывки *)
	(* Показать в панели сколько осталось до следующей промывки *)
	#415 regenByFT0102:FlowVolume(valueFT0102, setVolumeFS, resetVolumeFS)
	#416 totalAmountFS <= #415.out 1
	#417 OR(testValve.1, testValve.7)
	#418 FS020101:QueueManager(#415.out 2, #417, alarmFS.0, regimeFS.0, resetAlarms, #551.out 12, valveOpened.1, valveClosed.1, valveOpened.7, valveClosed.7, 45)
	#419 openValve.1 <= #418.out 2
	#420 closeValve.1 <= #418.out 3
	#421 alarmToOpenValve.1 <= #418.out 4
	#422 alarmToCloseValve.1 <= #418.out 5
	#423 openValve.7 <= #418.out 6
	#424 closeValve.7 <= #418.out 7
	#425 alarmToOpenValve.7 <= #418.out 8
	#426 alarmToCloseValve.7 <= #418.out 9
	#427 regeneratedFS.0 <= #418.out 10
	#428 failToRegenFS.0 <= #418.out 11
	#429 OR(testValve.2, testValve.8)
	#430 FS020102:QueueManager(#418.out 1, #429, alarmFS.1, regimeFS.1, resetAlarms, #551.out 12, valveOpened.2, valveClosed.2, valveOpened.8, valveClosed.8, 45)
	#431 openValve.2 <= #430.out 2
	#432 closeValve.2 <= #430.out 3
	#433 alarmToOpenValve.2 <= #430.out 4
	#434 alarmToCloseValve.2 <= #430.out 5
	#435 openValve.8 <= #430.out 6
	#436 closeValve.8 <= #430.out 7
	#437 alarmToOpenValve.8 <= #430.out 8
	#438 alarmToCloseValve.8 <= #430.out 9
	#439 regeneratedFS.1 <= #430.out 10
	#440 failToRegenFS.1 <= #430.out 11
	#441 OR(testValve.3, testValve.9)
	#442 FS020103:QueueManager(#430.out 1, #441, alarmFS.2, regimeFS.2, resetAlarms, #551.out 12, valveOpened.3, valveClosed.3, valveOpened.9, valveClosed.9, 45)
	#443 openValve.3 <= #442.out 2
	#444 closeValve.3 <= #442.out 3
	#445 alarmToOpenValve.3 <= #442.out 4
	#446 alarmToCloseValve.3 <= #442.out 5
	#447 openValve.9 <= #442.out 6
	#448 closeValve.9 <= #442.out 7
	#449 alarmToOpenValve.9 <= #442.out 8
	#450 alarmToCloseValve.9 <= #442.out 9
	#451 regeneratedFS.2 <= #442.out 10
	#452 failToRegenFS.2 <= #442.out 11
	#453 OR(testValve.4, testValve.10)
	#454 FS020104:QueueManager(#442.out 1, #453, alarmFS.3, regimeFS.3, resetAlarms, #551.out 12, valveOpened.4, valveClosed.4, valveOpened.10, valveClosed.10, 45)
	#455 openValve.4 <= #454.out 2
	#456 closeValve.4 <= #454.out 3
	#457 alarmToOpenValve.4 <= #454.out 4
	#458 alarmToCloseValve.4 <= #454.out 5
	#459 openValve.10 <= #454.out 6
	#460 closeValve.10 <= #454.out 7
	#461 alarmToOpenValve.10 <= #454.out 8
	#462 alarmToCloseValve.10 <= #454.out 9
	#463 regeneratedFS.3 <= #454.out 10
	#464 failToRegenFS.3 <= #454.out 11
	#465 OR(testValve.5, testValve.11)
	#466 FS020105:QueueManager(#454.out 1, #465, alarmFS.4, regimeFS.4, resetAlarms, #551.out 12, valveOpened.5, valveClosed.5, valveOpened.11, valveClosed.11, 45)
	#467 openValve.5 <= #466.out 2
	#468 closeValve.5 <= #466.out 3
	#469 alarmToOpenValve.5 <= #466.out 4
	#470 alarmToCloseValve.5 <= #466.out 5
	#471 openValve.11 <= #466.out 6
	#472 closeValve.11 <= #466.out 7
	#473 alarmToOpenValve.11 <= #466.out 8
	#474 alarmToCloseValve.11 <= #466.out 9
	#475 regeneratedFS.4 <= #466.out 10
	#476 failToRegenFS.4 <= #466.out 11
	#477 OR(testValve.6, testValve.12)
	#478 FS020106:QueueManager(#466.out 1, #477, alarmFS.5, regimeFS.5, resetAlarms, #551.out 12, valveOpened.6, valveClosed.6, valveOpened.12, valveClosed.12, 45)
	#479 openValve.6 <= #478.out 2
	#480 closeValve.6 <= #478.out 3
	#481 alarmToOpenValve.6 <= #478.out 4
	#482 alarmToCloseValve.6 <= #478.out 5
	#483 openValve.12 <= #478.out 6
	#484 closeValve.12 <= #478.out 7
	#485 alarmToOpenValve.12 <= #478.out 8
	#486 alarmToCloseValve.12 <= #478.out 9
	#487 regeneratedFS.5 <= #478.out 10
	#488 failToRegenFS.5 <= #478.out 11
	#489 setRegimeFS.0 <= #418.out 13
	#490 OR(testValve.13, testValve.19)
	#491 FS020201:QueueManager(#478.out 1, #490, alarmFS.6, regimeFS.6, resetAlarms, #551.out 12, valveOpened.13, valveClosed.13, valveOpened.19, valveClosed.19, 45)
	#492 openValve.13 <= #491.out 2
	#493 closeValve.13 <= #491.out 3
	#494 alarmToOpenValve.13 <= #491.out 4
	#495 alarmToCloseValve.13 <= #491.out 5
	#496 openValve.19 <= #491.out 6
	#497 closeValve.19 <= #491.out 7
	#498 alarmToOpenValve.19 <= #491.out 8
	#499 alarmToCloseValve.19 <= #491.out 9
	#500 regeneratedFS.6 <= #491.out 10
	#501 failToRegenFS.6 <= #491.out 11
	#502 OR(testValve.14, testValve.20)
	#503 FS020202:QueueManager(#491.out 1, #502, alarmFS.7, regimeFS.7, resetAlarms, #551.out 12, valveOpened.14, valveClosed.14, valveOpened.20, valveClosed.20, 45)
	#504 openValve.14 <= #503.out 2
	#505 closeValve.14 <= #503.out 3
	#506 alarmToOpenValve.14 <= #503.out 4
	#507 alarmToCloseValve.14 <= #503.out 5
	#508 openValve.20 <= #503.out 6
	#509 closeValve.20 <= #503.out 7
	#510 alarmToOpenValve.20 <= #503.out 8
	#511 alarmToCloseValve.20 <= #503.out 9
	#512 regeneratedFS.7 <= #503.out 10
	#513 failToRegenFS.7 <= #503.out 11
	#514 OR(testValve.15, testValve.21)
	#515 FS020203:QueueManager(#503.out 1, #514, alarmFS.8, regimeFS.8, resetAlarms, #551.out 12, valveOpened.15, valveClosed.15, valveOpened.21, valveClosed.21, 45)
	#516 openValve.15 <= #515.out 2
	#517 closeValve.15 <= #515.out 3
	#518 alarmToOpenValve.15 <= #515.out 4
	#519 alarmToCloseValve.15 <= #515.out 5
	#520 openValve.21 <= #515.out 6
	#521 closeValve.21 <= #515.out 7
	#522 alarmToOpenValve.21 <= #515.out 8
	#523 alarmToCloseValve.21 <= #515.out 9
	#524 regeneratedFS.8 <= #515.out 10
	#525 failToRegenFS.8 <= #515.out 11
	#526 OR(testValve.16, testValve.22)
	#527 FS020204:QueueManager(#515.out 1, #526, alarmFS.9, regimeFS.9, resetAlarms, #551.out 12, valveOpened.16, valveClosed.16, valveOpened.22, valveClosed.22, 45)
	#528 openValve.16 <= #527.out 2
	#529 closeValve.16 <= #527.out 3
	#530 alarmToOpenValve.16 <= #527.out 4
	#531 alarmToCloseValve.16 <= #527.out 5
	#532 openValve.22 <= #527.out 6
	#533 closeValve.22 <= #527.out 7
	#534 alarmToOpenValve.22 <= #527.out 8
	#535 alarmToCloseValve.22 <= #527.out 9
	#536 regeneratedFS.9 <= #527.out 10
	#537 failToRegenFS.9 <= #527.out 11
	#538 OR(testValve.17, testValve.23)
	#539 FS020205:QueueManager(#527.out 1, #538, alarmFS.10, regimeFS.10, resetAlarms, #551.out 12, valveOpened.17, valveClosed.17, valveOpened.23, valveClosed.23, 45)
	#540 openValve.17 <= #539.out 2
	#541 closeValve.17 <= #539.out 3
	#542 alarmToOpenValve.17 <= #539.out 4
	#543 alarmToCloseValve.17 <= #539.out 5
	#544 openValve.23 <= #539.out 6
	#545 closeValve.23 <= #539.out 7
	#546 alarmToOpenValve.23 <= #539.out 8
	#547 alarmToCloseValve.23 <= #539.out 9
	#548 regeneratedFS.10 <= #539.out 10
	#549 failToRegenFS.10 <= #539.out 11
	#550 OR(testValve.18, testValve.24)
	#551 FS020206:QueueManager(#539.out 1, #550, alarmFS.11, regimeFS.11, resetAlarms, #551.out 12, valveOpened.18, valveClosed.18, valveOpened.24, valveClosed.24, 45)
	#552 openValve.18 <= #551.out 2
	#553 closeValve.18 <= #551.out 3
	#554 alarmToOpenValve.18 <= #551.out 4
	#555 alarmToCloseValve.18 <= #551.out 5
	#556 openValve.24 <= #551.out 6
	#557 closeValve.24 <= #551.out 7
	#558 alarmToOpenValve.24 <= #551.out 8
	#559 alarmToCloseValve.24 <= #551.out 9
	#560 regeneratedFS.11 <= #551.out 10
	#561 failToRegenFS.11 <= #551.out 11
	#562 SUB(setVolumeFS, totalAmountFS)
	#563 toNextRegen <= #562
	#564 setRegimeFS.1 <= #430.out 13
	#565 setRegimeFS.2 <= #442.out 13
	#566 setRegimeFS.3 <= #454.out 13
	#567 setRegimeFS.4 <= #466.out 13
	#568 setRegimeFS.5 <= #478.out 13
	#569 setRegimeFS.6 <= #491.out 13
	#570 setRegimeFS.7 <= #503.out 13
	#571 setRegimeFS.8 <= #515.out 13
	#572 setRegimeFS.9 <= #527.out 13
	#573 setRegimeFS.10 <= #539.out 13
	#574 setRegimeFS.11 <= #551.out 13
END_MACRO
#575 MACRO Сигналы управления заслонками()
	(* КШЭ04.01 *)
	(* ЗДЭ03.02 *)
	(* ЗДЭ03.01 *)
	(* ЗДЭ02.25 *)
	(* ЗДЭ02.24 *)
	(* ЗДЭ02.23 *)
	(* ЗДЭ02.22 *)
	(* ЗДЭ02.21 *)
	(* ЗДЭ02.20 *)
	(* ЗДЭ02.19 *)
	(* ЗДЭ02.18 *)
	(* ЗДЭ02.17 *)
	(* ЗДЭ02.16 *)
	(* ЗДЭ02.15 *)
	(* ЗДЭ02.14 *)
	(* ЗДЭ02.13 *)
	(* ЗДЭ02.12 *)
	(* ЗДЭ02.11 *)
	(* ЗДЭ02.10 *)
	(* ЗДЭ02.09 *)
	(* ЗДЭ02.08 *)
	(* ЗДЭ02.07 *)
	(* ЗДЭ02.06 *)
	(* ЗДЭ02.05 *)
	(* ЗДЭ02.04 *)
	(* ЗДЭ02.03 *)
	(* ЗДЭ02.02 *)
	(* ЗДЭ02.01 *)
	(* ЗДЭ01.01 *)
	(* Сигналы управления заслонками *)
	(* Статус - заслонка закрыта *)
	(* Статус - заслонка открыта *)
	(* Закрыть заслонку *)
	(* Открыть заслонку *)
	#576 DD2_1_DO.0 <= openValve.0
	#577 DD2_1_DO.1 <= closeValve.0
	#578 DD2_1_DO.2 <= openValve.1
	#579 DD2_1_DO.3 <= closeValve.1
	#580 DD2_1_DO.4 <= openValve.2
	#581 DD2_1_DO.5 <= closeValve.2
	#582 DD2_1_DO.6 <= openValve.3
	#583 DD2_1_DO.7 <= closeValve.3
	#584 DD2_1_DO.8 <= openValve.4
	#585 DD2_1_DO.9 <= closeValve.4
	#586 DD2_1_DO.10 <= openValve.5
	#587 DD2_1_DO.11 <= closeValve.5
	#588 DD2_1_DO.12 <= openValve.6
	#589 DD2_1_DO.13 <= closeValve.6
	#590 DD2_1_DO.14 <= openValve.7
	#591 DD2_1_DO.15 <= closeValve.7
	#592 DD2_1_DO.16 <= openValve.8
	#593 DD2_1_DO.17 <= closeValve.8
	#594 DD2_1_DO.18 <= openValve.9
	#595 DD2_1_DO.19 <= closeValve.9
	#596 DD2_1_DO.20 <= openValve.10
	#597 DD2_1_DO.21 <= closeValve.10
	#598 DD2_1_DO.22 <= openValve.11
	#599 DD2_1_DO.23 <= closeValve.11
	#600 DD2_1_DO.24 <= openValve.12
	#601 DD2_1_DO.25 <= closeValve.12
	#602 DD2_1_DO.26 <= openValve.13
	#603 DD2_1_DO.27 <= closeValve.13
	#604 DD2_1_DO.28 <= openValve.14
	#605 DD2_1_DO.29 <= closeValve.14
	#606 DD2_1_DO.30 <= openValve.15
	#607 DD2_1_DO.31 <= closeValve.15
	#608 DD2_2_DO.0 <= openValve.16
	#609 DD2_2_DO.1 <= closeValve.16
	#610 DD2_2_DO.2 <= openValve.17
	#611 DD2_2_DO.3 <= closeValve.17
	#612 DD2_2_DO.4 <= openValve.18
	#613 DD2_2_DO.5 <= closeValve.18
	#614 DD2_2_DO.6 <= openValve.19
	#615 DD2_2_DO.7 <= closeValve.19
	#616 DD2_2_DO.8 <= openValve.20
	#617 DD2_2_DO.9 <= closeValve.20
	#618 DD2_2_DO.10 <= openValve.21
	#619 DD2_2_DO.11 <= closeValve.21
	#620 DD2_2_DO.12 <= openValve.22
	#621 DD2_2_DO.13 <= closeValve.22
	#622 DD2_2_DO.14 <= openValve.23
	#623 DD2_2_DO.15 <= closeValve.23
	#624 DD2_2_DO.16 <= openValve.24
	#625 DD2_2_DO.17 <= closeValve.24
	#626 DD2_2_DO.18 <= openValve.25
	#627 DD2_2_DO.19 <= closeValve.25
	#628 DD2_2_DO.20 <= openValve.26
	#629 DD2_2_DO.21 <= closeValve.26
	#630 DD2_2_DO.22 <= openValve.27
	#631 DD2_2_DO.23 <= closeValve.27
	#632 DD2_2_DO.24 <= openValve.28
	#633 DD2_2_DO.25 <= closeValve.28
	#634 openRS0:RS(SET: DD2_4_DI.1, RESET1: closeValve.0)
	#635 valveOpened.0 <= #634.Q1
	#636 closeRS0:RS(SET: DD2_4_DI.2, RESET1: openValve.0)
	#637 valveClosed.0 <= #636.Q1
	#638 openRS1:RS(SET: DD2_4_DI.3, RESET1: closeValve.1)
	#639 valveOpened.1 <= #638.Q1
	#640 closeRS1:RS(SET: DD2_4_DI.4, RESET1: openValve.1)
	#641 valveClosed.1 <= #640.Q1
	#642 openRS2:RS(SET: DD2_4_DI.5, RESET1: closeValve.2)
	#643 valveOpened.2 <= #642.Q1
	#644 closeRS2:RS(SET: DD2_4_DI.6, RESET1: openValve.2)
	#645 valveClosed.2 <= #644.Q1
	#646 openRS3:RS(SET: DD2_4_DI.7, RESET1: closeValve.3)
	#647 valveOpened.3 <= #646.Q1
	#648 closeRS3:RS(SET: DD2_4_DI.8, RESET1: openValve.3)
	#649 valveClosed.3 <= #648.Q1
	#650 openRS4:RS(SET: DD2_4_DI.9, RESET1: closeValve.4)
	#651 valveOpened.4 <= #650.Q1
	#652 closeRS4:RS(SET: DD2_4_DI.10, RESET1: openValve.4)
	#653 valveClosed.4 <= #652.Q1
	#654 openRS5:RS(SET: DD2_4_DI.11, RESET1: closeValve.5)
	#655 valveOpened.5 <= #654.Q1
	#656 closeRS5:RS(SET: DD2_4_DI.12, RESET1: openValve.5)
	#657 valveClosed.5 <= #656.Q1
	#658 openRS6:RS(SET: DD2_4_DI.13, RESET1: closeValve.6)
	#659 valveOpened.6 <= #658.Q1
	#660 closeRS6:RS(SET: DD2_4_DI.14, RESET1: openValve.6)
	#661 valveClosed.6 <= #660.Q1
	#662 openRS7:RS(SET: DD2_4_DI.15, RESET1: closeValve.7)
	#663 valveOpened.7 <= #662.Q1
	#664 closeRS7:RS(SET: DD2_4_DI.16, RESET1: openValve.7)
	#665 valveClosed.7 <= #664.Q1
	#666 openRS8:RS(SET: DD2_4_DI.17, RESET1: closeValve.8)
	#667 valveOpened.8 <= #666.Q1
	#668 closeRS8:RS(SET: DD2_4_DI.18, RESET1: openValve.8)
	#669 valveClosed.8 <= #668.Q1
	#670 openRS9:RS(SET: DD2_4_DI.19, RESET1: closeValve.9)
	#671 valveOpened.9 <= #670.Q1
	#672 closeRS9:RS(SET: DD2_4_DI.20, RESET1: openValve.9)
	#673 valveClosed.9 <= #672.Q1
	#674 openRS10:RS(SET: DD2_4_DI.21, RESET1: closeValve.10)
	#675 valveOpened.10 <= #674.Q1
	#676 closeRS10:RS(SET: DD2_4_DI.22, RESET1: openValve.10)
	#677 valveClosed.10 <= #676.Q1
	#678 openRS11:RS(SET: DD2_4_DI.23, RESET1: closeValve.11)
	#679 valveOpened.11 <= #678.Q1
	#680 closeRS11:RS(SET: DD2_4_DI.24, RESET1: openValve.11)
	#681 valveClosed.11 <= #680.Q1
	#682 openRS12:RS(SET: DD2_4_DI.25, RESET1: closeValve.12)
	#683 valveOpened.12 <= #682.Q1
	#684 closeRS12:RS(SET: DD2_4_DI.26, RESET1: openValve.12)
	#685 valveClosed.12 <= #684.Q1
	#686 openRS13:RS(SET: DD2_4_DI.27, RESET1: closeValve.13)
	#687 valveOpened.13 <= #686.Q1
	#688 closeRS13:RS(SET: DD2_4_DI.28, RESET1: openValve.13)
	#689 valveClosed.13 <= #688.Q1
	#690 openRS14:RS(SET: DD2_4_DI.29, RESET1: closeValve.14)
	#691 valveOpened.14 <= #690.Q1
	#692 closeRS14:RS(SET: DD2_4_DI.30, RESET1: openValve.14)
	#693 valveClosed.14 <= #692.Q1
	#694 openRS15:RS(SET: DD2_4_DI.31, RESET1: closeValve.15)
	#695 valveOpened.15 <= #694.Q1
	#696 closeRS15:RS(SET: DD2_5_DI.0, RESET1: openValve.15)
	#697 valveClosed.15 <= #696.Q1
	#698 openRS16:RS(SET: DD2_5_DI.1, RESET1: closeValve.16)
	#699 valveOpened.16 <= #698.Q1
	#700 closeRS16:RS(SET: DD2_5_DI.2, RESET1: openValve.16)
	#701 valveClosed.16 <= #700.Q1
	#702 openRS17:RS(SET: DD2_5_DI.3, RESET1: closeValve.17)
	#703 valveOpened.17 <= #702.Q1
	#704 closeRS17:RS(SET: DD2_5_DI.4, RESET1: openValve.17)
	#705 valveClosed.17 <= #704.Q1
	#706 openRS18:RS(SET: DD2_5_DI.5, RESET1: closeValve.18)
	#707 valveOpened.18 <= #706.Q1
	#708 closeRS18:RS(SET: DD2_5_DI.6, RESET1: openValve.18)
	#709 valveClosed.18 <= #708.Q1
	#710 openRS19:RS(SET: DD2_5_DI.7, RESET1: closeValve.19)
	#711 valveOpened.19 <= #710.Q1
	#712 closeRS19:RS(SET: DD2_5_DI.8, RESET1: openValve.19)
	#713 valveClosed.19 <= #712.Q1
	#714 openRS20:RS(SET: DD2_5_DI.9, RESET1: closeValve.20)
	#715 valveOpened.20 <= #714.Q1
	#716 closeRS20:RS(SET: DD2_5_DI.10, RESET1: openValve.20)
	#717 valveClosed.20 <= #716.Q1
	#718 openRS21:RS(SET: DD2_5_DI.11, RESET1: closeValve.21)
	#719 valveOpened.21 <= #718.Q1
	#720 closeRS21:RS(SET: DD2_5_DI.12, RESET1: openValve.21)
	#721 valveClosed.21 <= #720.Q1
	#722 openRS22:RS(SET: DD2_5_DI.13, RESET1: closeValve.22)
	#723 valveOpened.22 <= #722.Q1
	#724 closeRS22:RS(SET: DD2_5_DI.14, RESET1: openValve.22)
	#725 valveClosed.22 <= #724.Q1
	#726 openRS23:RS(SET: DD2_5_DI.15, RESET1: closeValve.23)
	#727 valveOpened.23 <= #726.Q1
	#728 closeRS23:RS(SET: DD2_5_DI.16, RESET1: openValve.23)
	#729 valveClosed.23 <= #728.Q1
	#730 openRS24:RS(SET: DD2_5_DI.17, RESET1: closeValve.24)
	#731 valveOpened.24 <= #730.Q1
	#732 closeRS24:RS(SET: DD2_5_DI.18, RESET1: openValve.24)
	#733 valveClosed.24 <= #732.Q1
	#734 openRS25:RS(SET: DD2_5_DI.19, RESET1: closeValve.25)
	#735 valveOpened.25 <= #734.Q1
	#736 closeRS25:RS(SET: DD2_5_DI.20, RESET1: openValve.25)
	#737 valveClosed.25 <= #736.Q1
	#738 openRS26:RS(SET: DD2_5_DI.21, RESET1: closeValve.26)
	#739 valveOpened.26 <= #738.Q1
	#740 closeRS26:RS(SET: DD2_5_DI.22, RESET1: openValve.26)
	#741 valveClosed.26 <= #740.Q1
	#742 openRS27:RS(SET: DD2_5_DI.23, RESET1: closeValve.27)
	#743 valveOpened.27 <= #742.Q1
	#744 closeRS27:RS(SET: DD2_5_DI.24, RESET1: openValve.27)
	#745 valveClosed.27 <= #744.Q1
	#746 openRS28:RS(SET: DD2_5_DI.25, RESET1: closeValve.28)
	#747 valveOpened.28 <= #746.Q1
	#748 closeRS28:RS(SET: DD2_5_DI.26, RESET1: openValve.28)
	#749 valveClosed.28 <= #748.Q1
END_MACRO
#750 MACRO Блок контроля и управления УФО03.01()
	(* Если расход по FT01.02 больше / или равен 10 куб.метров/час, / то запускаем УФО. *)
	(* Пуск УФО03.01/01 *)
	(* Cтоп УФО03.01/01 *)
	(* Авария УФО03.01/01 *)
	(* Пуск УФО03.01/02 *)
	(* Cтоп УФО03.01/02 *)
	(* Авария УФО03.01/02 *)
	(* Блок контроля и управления УФО03.01 *)
	#751 GE(valueFT0102, 10)
	#752 setWordUFO0301.0 <= #751
	#753 UFO0301manager:RichTwoPumpManager(setWordUFO0301.0, setWordUFO0301.1, setWordUFO0301.2, setWordUFO0301.3, setWordUFO0301.4, setWordUFO0301.5, setWordUFO0301.6, setWordUFO0301.7, setWordUFO0301.8, setWordUFO0301.9, setWordUFO0301.10, setWordUFO0301.11, resetAlarms, -, statusUFO030101alarm, statusUFO030102alarm)
	#754 statWordUFO0301.1 <= #753.out 1
	#755 statWordUFO0301.2 <= #753.out 2
	#756 statWordUFO0301.3 <= #753.out 3
	#757 statWordUFO0301.4 <= #753.out 4
	#758 counterUFO030101 <= #753.out 5
	#759 counterUFO030102 <= #753.out 6
	#760 daysUFO030101 <= #753.out 7
	#761 statusStart.7 <= #753.out 15
	#762 hoursUFO030101 <= #753.out 8
	#763 UFO030101start <= #753.out 15
	#764 minutesUFO030101 <= #753.out 9
	#765 UFO030101stop <= NOT #753.out 15
	#766 secondsUFO030101 <= #753.out 10
	#767 daysUFO030102 <= #753.out 11
	#768 hoursUFO030102 <= #753.out 12
	#769 minutesUFO030102 <= #753.out 13
	#770 secondsUFO030102 <= #753.out 14
	#771 statWordUFO0301.5 <= #753.out 19
	#772 statusStart.8 <= #753.out 16
	#773 statWordUFO0301.6 <= #753.out 20
	#774 UFO030102start <= #753.out 16
	#775 UFO030102stop <= NOT #753.out 16
	#776 OR(#753.out 15, testValve.26)
	#777 ZDE0301:SimpleValve(#776, NOT #776, valveOpened.26, valveClosed.26, resetAlarms, 45)
	#778 openValve.26 <= #777.out 1
	#779 closeValve.26 <= #777.out 2
	#780 alarmToOpenValve.26 <= #777.out 3
	#781 alarmToCloseValve.26 <= #777.out 4
	#782 OR(#753.out 16, testValve.27)
	#783 ZDE0302:SimpleValve(#782, NOT #782, valveOpened.27, valveClosed.27, resetAlarms, 45)
	#784 openValve.27 <= #783.out 1
	#785 closeValve.27 <= #783.out 2
	#786 alarmToOpenValve.27 <= #783.out 3
	#787 alarmToCloseValve.27 <= #783.out 4
END_MACRO
#788 MACRO передача сигналов уровней емкостей в панель()
	(* LS01.04 Сухой ход Н01.05 / 0 = сухой ход *)
	(* LS02.03 Сухой ход Н02.04 / 0 = сухой ход *)
	(* LS04.01 Верхний уровень ПР04.03 / 1 = верх.уровень, пуск Н04.04 *)
	(* LS04.02 Сухой ход Н04.04 / 0 = сухой ход *)
	(* LS08.02 Сухой ход НД08.03/01 / 0 = сухой ход *)
	(* LS08.03 Сухой ход НД08.03/02 / 0 = сухой ход *)
	(* LS01.01 Сухой ход Н04.01 (Защита ФПК) / 0 = сухой ход *)
	(* LSA01.02 Перелив ОГМ01.04 / 0 = перелив *)
	(* LS01.03 Рабочий верхний уровень ОГМ01.04 / 1 = верх. уровень, пуск Н01.05 *)
	(* LSA02.01 Перелив РЧВ02.03 / 0 = перелив *)
	(* LS02.02 Рабочий верхний уровень РЧВ02.03 / 1 = наполнение, открыть ЗДЭ02.25 *)
	(* Сигнал уровня осадка LES01.01 / 1 = пора обезвоживать *)
	#789 levelStatus.0 <= NOT DD1_2_DI.30
	#790 levelStatus.1 <= DD1_2_DI.31
	#791 levelStatus.2 <= NOT DD1_2_DI.5
	#792 levelStatus.3 <= NOT DD1_3_DI.0
	#793 levelStatus.4 <= DD1_3_DI.1
	#794 levelStatus.5 <= NOT DD1_2_DI.8
	#795 levelStatus.6 <= DD1_2_DI.9
	#796 levelStatus.7 <= NOT DD1_2_DI.10
	#797 levelStatus.8 <= NOT DD1_2_DI.27
	#798 levelStatus.9 <= NOT DD1_2_DI.28
	#799 levelStatus.10 <= NOT DD1_2_DI.29
	#800 levelStatus.11 <= DD2_6_DI.23
END_MACRO
#801 MACRO Контроль температуры в помещении()
	(* Контроль нахождения температуры в помещении / в заданном диапазоне. *)
	#802 GT(valueTemperature, setMaxTemperature)
	#803 alarmTemperatureHigh <= #802
	#804 LT(valueTemperature, setMinTemperature)
	#805 alarmTemperatureLow <= #804
END_MACRO
#806 MACRO Блок управления заслонкой на входе в станцию (ЗДЭ01.01)()
	(* авария УФО03.01/01 *)
	(* Блок управления заслонкой на входе в станцию (ЗДЭ01.01) *)
	(* авария УФО03.01/02 *)
	(* Перелив ОГМ01.04 *)
	#807 AND(statWordUFO0301.5, statWordUFO0301.6)
	#808 OR(testValve.0, DD1_2_DI.30, #807)
	#809 ZDE0101:SimpleValve(NOT #808, #808, valveOpened.0, valveClosed.0, resetAlarms, 45)
	#810 openValve.0 <= #809.out 1
	#811 closeValve.0 <= #809.out 2
	#812 alarmToOpenValve.0 <= #809.out 3
	#813 alarmToCloseValve.0 <= #809.out 4
END_MACRO
#814 MACRO счетчик очищенных стоков (FQS03.01)()
	(* Импульсный счетчик очищенных стоков. *)
	#815 CounterFQS0301impulses:ImpulsFlowCounter(DD2_7_DI0, impulsValueFQS0301, resetCounterFQS0301, correctionValueFQS0301, addCorrectionFQS0301, deleteCorrectionFQS0301)
	#816 totalAmountFQS0301 <= #815.out 2
END_MACRO
#817 MACRO Диспетчеризация()
	#818 remFT0101value <= valueFT0101
	#819 remFQS0301totalAmount <= totalAmountFQS0301
	#820 remTemperatureValue <= valueTemperature
	#821 remStatusN010501started <= statusStart.0
	#822 remStatusN010502started <= statusStart.1
	#823 remStatusUFO030101started <= statusStart.7
	#824 remStatusUFO030102started <= statusStart.8
	#825 remAlarm <= alarm
	#826 OR(statWordN0105.5, powerAlarmN0105)
	#827 remN010501alarm <= #826
	#828 OR(powerAlarmN0105, statWordN0105.6)
	#829 remN010502alarm <= #828
	#830 remFPKalarm <= alarmFPK
	#831 remUFO030101alarm <= statWordUFO0301.5
	#832 remUFO030102alarm <= statWordUFO0301.6
	#833 remAlarmOOGM0104overload <= levelStatus.0
	#834 remAlarmRCHV0203overload <= levelStatus.3
END_MACRO
#835 MACRO чтение переменных из панели()
	#836 impulsValueFQS0301 <= impulsValueFQS0301PAN
	#837 timeToWorkFPK <= timeToWorkFPKPAN
	#838 maxPressureValueFPK <= maxPressureValueFPKPAN
	#839 ND0502setMaxDosVal <= ND0502setMaxDosValPAN
	#840 ND0502setKoefProp <= ND0502setKoefPropPAN
	#841 ND0602setMaxDosVal <= ND0602setMaxDosValPAN
	#842 ND0602setKoefProp <= ND0602setKoefPropPAN
	#843 ND0603setMaxDosVal <= ND0603setMaxDosValPAN
	#844 ND0603setKoefProp <= ND0603setKoefPropPAN
	#845 ND0703pHsetValue <= ND0703pHsetValuePAN
	#846 REAL_TO_WORD(ND0703YoutManualPAN)
	#847 ND0703YoutManual <= #846
	#848 ND0803setMaxDosVal <= ND0803setMaxDosValPAN
	#849 ND0803setKoefProp <= ND0803setKoefPropPAN
	#850 REAL_TO_WORD(ND0804doseValuePAN)
	#851 ND0804doseValue <= #850
	#852 N0105flowSetValue <= N0105flowSetValuePAN
	#853 REAL_TO_WORD(N0105YoutManualPAN)
	#854 N0105YoutManual <= #853
	#855 setVolumeFS <= setVolumeFSPAN
	#856 setMinTemperature <= setMinTemperaturePAN
	#857 setMaxTemperature <= setMaxTemperaturePAN
	#858 correctionValueFQS0301 <= correctionValueFQS0301PAN
	#859 setWordND0502 <= setWordND0502PAN
	#860 setWordND0602 <= setWordND0602PAN
	#861 setWordND0603 <= setWordND0603PAN
	#862 setWordND0703 <= setWordND0703PAN
	#863 setWordND0803 <= setWordND0803PAN
	#864 setWordN0105 <= setWordN0105PAN
	#865 setWordN0404 <= setWordN0404PAN
	#866 setWordUFO0301 <= setWordUFO0301PAN
	#867 setWordN0204 <= setWordN0204PAN
	#868 testValve <= testValvePAN
	#869 resetCounterFQS0301 <= resetCounterFQS0301PAN
	#870 addCorrectionFQS0301 <= addCorrectionFQS0301PAN
	#871 deleteCorrectionFQS0301 <= deleteCorrectionFQS0301PAN
	#872 ND0703YmanAuto <= ND0703YmanAutoPAN
	#873 N0105YmanAuto <= N0105YmanAutoPAN
	#874 resetVolumeFS <= resetVolumeFSPAN
	#875 N0105manStart <= N0105manStartPAN
	#876 N0105manStop <= N0105manStopPAN
	#877 N0204manStart <= N0204manStartPAN
	#878 N0204manStop <= N0204manStopPAN
	#879 N0404manStart <= N0404manStartPAN
	#880 N0404manStop <= N0404manStopPAN
	#881 resetAlarms <= resetAlarmsPAN
END_MACRO
#882 MACRO запись переменных в панель()
	#883 valueTemperaturePAN <= valueTemperature
	#884 minutesND060201PAN <= minutesND060201
	#885 secondsND070301PAN <= secondsND070301
	#886 hoursN010502PAN <= hoursN010502
	#887 secondsUFO030102PAN <= secondsUFO030102
	#888 statWordN0105PAN <= statWordN0105
	#889 powerAlarmRelay2PAN <= powerAlarmRelay2
	#890 valueFT0101PAN <= valueFT0101
	#891 secondsND060201PAN <= secondsND060201
	#892 daysND070302PAN <= daysND070302
	#893 minutesN010502PAN <= minutesN010502
	#894 counterN020401PAN <= counterN020401
	#895 statWordN0404PAN <= statWordN0404
	#896 notStartedFPKPAN <= notStartedFPK
	#897 valueFT0102PAN <= valueFT0102
	#898 daysND060202PAN <= daysND060202
	#899 hoursND070302PAN <= hoursND070302
	#900 secondsN010502PAN <= secondsN010502
	#901 counterN020402PAN <= counterN020402
	#902 statWordUFO0301PAN <= statWordUFO0301
	#903 alarmPLKnetworkPAN <= alarmPLKnetwork
	#904 valueFT0102PAN <= valueFT0102
	#905 hoursND060202PAN <= hoursND060202
	#906 minutesND070302PAN <= minutesND070302
	#907 counterN040401PAN <= counterN040401
	#908 daysN020401PAN <= daysN020401
	#909 statWordN0204PAN <= statWordN0204
	#910 valueQE0102PAN <= valueQE0102
	#911 hoursND060202PAN <= hoursND060202
	#912 secondsND070302PAN <= secondsND070302
	#913 counterN040402PAN <= counterN040402
	#914 hoursN020401PAN <= hoursN020401
	#915 alarmAIPAN <= alarmAI
	#916 valueFPKpressurePAN <= valueFPKpressure
	#917 minutesND060202PAN <= minutesND060202
	#918 counterND080301PAN <= counterND080301
	#919 daysN040401PAN <= daysN040401
	#920 minutesN020401PAN <= minutesN020401
	#921 alarmToOpenValvePAN <= alarmToOpenValve
	#922 totalAmountFQS0301PAN <= totalAmountFQS0301
	#923 secondsND060202PAN <= secondsND060202
	#924 counterND080302PAN <= counterND080302
	#925 hoursN040401PAN <= hoursN040401
	#926 secondsN020401PAN <= secondsN020401
	#927 alarmToCloseValvePAN <= alarmToCloseValve
	#928 toNextRegenPAN <= toNextRegen
	#929 counterND060301PAN <= counterND060301
	#930 daysND080301PAN <= daysND080301
	#931 minutesN040401PAN <= minutesN040401
	#932 daysN020402PAN <= daysN020402
	#933 alarmFSPAN <= alarmFS
	#934 counterND050201PAN <= counterND050201
	#935 counterND060302PAN <= counterND060302
	#936 hoursND080301PAN <= hoursND080301
	#937 secondsN040401PAN <= secondsN040401
	#938 hoursN020402PAN <= hoursN020402
	#939 failToRegenFSPAN <= failToRegenFS
	#940 counterND050202PAN <= counterND050201
	#941 daysND060301PAN <= daysND060301
	#942 minutesND080301PAN <= minutesND080301
	#943 daysN040402PAN <= daysN040402
	#944 minutesN020402PAN <= minutesN020402
	#945 needToCleanFPKPAN <= needToCleanFPK
	#946 daysND050201PAN <= daysND050201
	#947 hoursND060301PAN <= hoursND060301
	#948 secondsND080301PAN <= secondsND080301
	#949 hoursN040402PAN <= hoursN040402
	#950 secondsN020402PAN <= secondsN020402
	#951 readyFPKPAN <= readyFPK
	#952 hoursND050201PAN <= hoursND050201
	#953 minutesND060301PAN <= minutesND060301
	#954 daysND080302PAN <= daysND080302
	#955 minutesN040402PAN <= minutesN040402
	#956 statusNDstartPAN <= statusNDstart
	#957 alarmPAN <= alarm
	#958 minutesND050201PAN <= minutesND050201
	#959 secondsND060301PAN <= secondsND060301
	#960 hoursND080302PAN <= hoursND080302
	#961 secondsN040402PAN <= secondsN040402
	#962 statusStartPAN <= statusStart
	#963 alarmFPKPAN <= alarmFPK
	#964 secondsND050201PAN <= secondsND050201
	#965 daysND060302PAN <= daysND060302
	#966 minutesND080302PAN <= minutesND080302
	#967 counterUFO030101PAN <= counterUFO030101
	#968 valveOpenedPAN <= valveOpened
	#969 alarmTemperatureHighPAN <= alarmTemperatureHigh
	#970 daysND050202PAN <= daysND050202
	#971 hoursND060302PAN <= hoursND060302
	#972 secondsND080302PAN <= secondsND080302
	#973 counterUFO030102PAN <= counterUFO030102
	#974 regimeFSPAN <= regimeFS
	#975 alarmTemperatureLowPAN <= alarmTemperatureLow
	#976 hoursND050202PAN <= hoursND050202
	#977 minutesND060302PAN <= minutesND060302
	#978 counterN010501PAN <= counterN010501
	#979 daysUFO030101PAN <= daysUFO030101
	#980 levelStatusPAN <= levelStatus
	#981 powerAlarmN0105PAN <= powerAlarmN0105
	#982 minutesND050202PAN <= minutesND050202
	#983 secondsND060302PAN <= secondsND060302
	#984 counterN010502PAN <= counterN010502
	#985 hoursUFO030101PAN <= hoursUFO030101
	#986 valveClosedPAN <= valveClosed
	#987 alarmM0604PAN <= alarmM0604
	#988 secondsND050202PAN <= secondsND050202
	#989 counterND070301PAN <= counterND070301
	#990 daysN010501PAN <= daysN010501
	#991 minutesUFO030101PAN <= minutesUFO030101
	#992 statWordND0502PAN <= statWordND0502
	#993 alarmM0702PAN <= alarmM0702
	#994 counterND060201PAN <= counterND060201
	#995 counterND070302PAN <= counterND070302
	#996 hoursN010501PAN <= hoursN010501
	#997 secondsUFO030101PAN <= secondsUFO030101
	#998 statWordND0602PAN <= statWordND0602
	#999 alarmM0802PAN <= alarmM0802
	#1000 counterND060202PAN <= counterND060202
	#1001 daysND070301PAN <= daysND070301
	#1002 minutesN010501PAN <= minutesN010501
	#1003 daysUFO030102PAN <= daysUFO030102
	#1004 statWordND0603PAN <= statWordND0603
	#1005 powerAlarmFSPAN <= powerAlarmFS
	#1006 daysND060201PAN <= daysND060201
	#1007 hoursND070301PAN <= hoursND070301
	#1008 secondsN010501PAN <= secondsN010501
	#1009 hoursUFO030102PAN <= hoursUFO030102
	#1010 statWordND0703PAN <= statWordND0703
	#1011 powerAlarmKEMPAN <= powerAlarmKEM
	#1012 hoursND060201PAN <= hoursND060201
	#1013 minutesND070301PAN <= minutesND070301
	#1014 daysN010502PAN <= daysN010502
	#1015 minutesUFO030102PAN <= minutesUFO030102
	#1016 statWordND0803PAN <= statWordND0803
	#1017 powerAlarmRelay1PAN <= powerAlarmRelay1
END_MACRO
_END_CFC_
END_PROGRAM

(* POU StartStopVFD, CFC *)
FUNCTION_BLOCK StartStopVFD
VAR_INPUT
	startStop: BOOL;		(*1 = старт, 0 = стоп.*)
END_VAR
VAR_OUTPUT
	commandWord: WORD;		(*Командное слово в ЧРП.*)
END_VAR
VAR
END_VAR
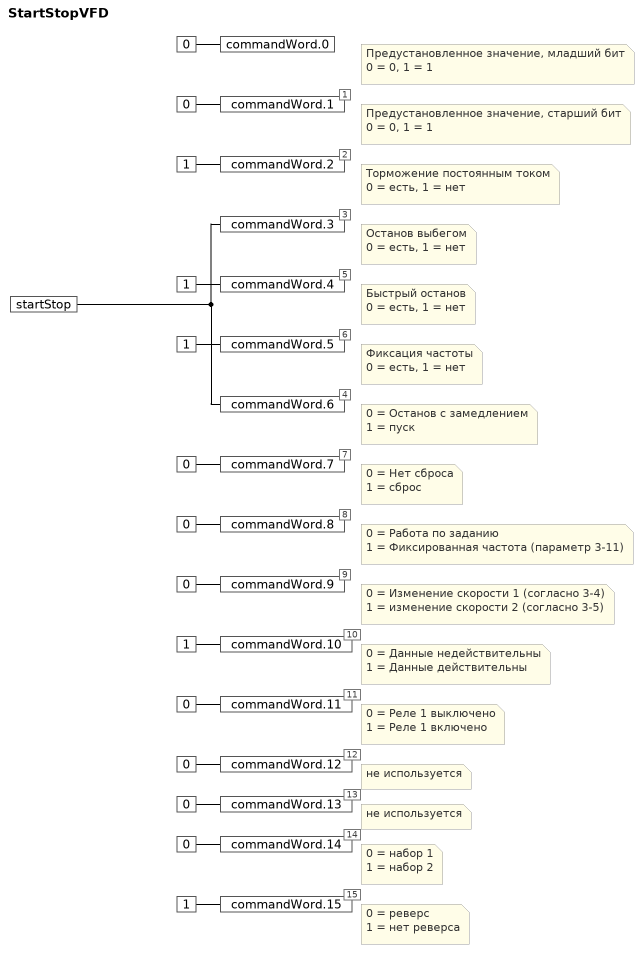
_CFC_ (* Continuous Function Chart, elements in execution order *)
(* 0 = реверс / 1 = нет реверса *)
(* 0 = набор 1 / 1 = набор 2 *)
(* не используется *)
(* не используется *)
(* 0 = Реле 1 выключено / 1 = Реле 1 включено *)
(* 0 = Данные недействительны / 1 = Данные действительны *)
(* 0 = Изменение скорости 1 (согласно 3-4) / 1 = изменение скорости 2 (согласно 3-5) *)
(* 0 = Работа по заданию / 1 = Фиксированная частота (параметр 3-11) *)
(* 0 = Нет сброса / 1 = сброс *)
(* 0 = Останов с замедлением / 1 = пуск *)
(* Фиксация частоты / 0 = есть, 1 = нет *)
(* Быстрый останов / 0 = есть, 1 = нет *)
(* Останов выбегом / 0 = есть, 1 = нет *)
(* Торможение постоянным током / 0 = есть, 1 = нет *)
(* Предустановленное значение, старший бит / 0 = 0, 1 = 1 *)
(* Предустановленное значение, младший бит / 0 = 0, 1 = 1 *)
#0 commandWord.0 <= 0
#1 commandWord.1 <= 0
#2 commandWord.2 <= 1
#3 commandWord.3 <= startStop
#4 commandWord.6 <= startStop
#5 commandWord.4 <= 1
#6 commandWord.5 <= 1
#7 commandWord.7 <= 0
#8 commandWord.8 <= 0
#9 commandWord.9 <= 0
#10 commandWord.10 <= 1
#11 commandWord.11 <= 0
#12 commandWord.12 <= 0
#13 commandWord.13 <= 0
#14 commandWord.14 <= 0
#15 commandWord.15 <= 1
_END_CFC_
(* the same logic as Structured Text *)
(* 0 = реверс / 1 = нет реверса *)
(* 0 = набор 1 / 1 = набор 2 *)
(* не используется *)
(* не используется *)
(* 0 = Реле 1 выключено / 1 = Реле 1 включено *)
(* 0 = Данные недействительны / 1 = Данные действительны *)
(* 0 = Изменение скорости 1 (согласно 3-4) / 1 = изменение скорости 2 (согласно 3-5) *)
(* 0 = Работа по заданию / 1 = Фиксированная частота (параметр 3-11) *)
(* 0 = Нет сброса / 1 = сброс *)
(* 0 = Останов с замедлением / 1 = пуск *)
(* Фиксация частоты / 0 = есть, 1 = нет *)
(* Быстрый останов / 0 = есть, 1 = нет *)
(* Останов выбегом / 0 = есть, 1 = нет *)
(* Торможение постоянным током / 0 = есть, 1 = нет *)
(* Предустановленное значение, старший бит / 0 = 0, 1 = 1 *)
(* Предустановленное значение, младший бит / 0 = 0, 1 = 1 *)
commandWord.0 := 0;
commandWord.1 := 0;
commandWord.2 := 1;
commandWord.3 := startStop;
commandWord.6 := startStop;
commandWord.4 := 1;
commandWord.5 := 1;
commandWord.7 := 0;
commandWord.8 := 0;
commandWord.9 := 0;
commandWord.10 := 1;
commandWord.11 := 0;
commandWord.12 := 0;
commandWord.13 := 0;
commandWord.14 := 0;
commandWord.15 := 1;
END_FUNCTION_BLOCK
